	(*Inverter comm error*)	AddError[w_Index](
			b_ErrorTrig			:= Get.ui_InverterCommStatus <>0 AND Get.ui_InverterCommStatus <15, //general warning from inverter
			out_ST_Error			:= a_ActiveEvents[w_Index],
			w_ErrorID					:= 66 ,
			s_Message				:= 'inverter communication error',
			e_sev					:= eSeverity.Quickshutdown
			);
		IF AddError[w_Index].b_out THEN by_errCt := by_errCt + 1; END_IF;
		w_Index := w_Index +1;
		
	(*Inverter temp throttling active*)	AddError[w_Index](
			b_ErrorTrig			:= get.Events.b_TempThrottlingActive, //general warning from inverter
			out_ST_Error			:= a_ActiveEvents[w_Index],
			w_ErrorID					:= 67 ,
			s_Message				:= 'temperature throttling active',
			e_sev					:= eSeverity.Warning,
			b_AutoClear			:= TRUE,
			);
		IF AddError[w_Index].b_out THEN by_warnCt := by_warnCt + 1; END_IF;
		w_Index := w_Index +1;
		
	(*Inverter current throttling active*)	AddError[w_Index](
			b_ErrorTrig			:= get.Events.b_CurrThrottlingActive, //general warning from inverter
			out_ST_Error			:= a_ActiveEvents[w_Index],
			w_ErrorID					:= 68 ,
			s_Message				:= 'Current throttling active',
			e_sev					:= eSeverity.Warning,
			b_AutoClear			:= TRUE,
			);
		IF AddError[w_Index].b_out THEN by_warnCt := by_warnCt + 1; END_IF;
		w_Index := w_Index +1;
		
		(*Inverter current throttling active*)	AddError[w_Index](
			b_ErrorTrig			:= get.StatusWord.b_Fault, //general warning from inverter
			out_ST_Error			:= a_ActiveEvents[w_Index],
			w_ErrorID					:= 69,
			s_Message				:= 'General fault',
			e_sev					:= eSeverity.Quickshutdown,
			);
		IF AddError[w_Index].b_out THEN by_errCt := by_errCt + 1; END_IF;
		w_Index := w_Index +1;
		
		(*UVR fault*)			AddError[w_Index](
			b_ErrorTrig				:= Get.Events.b_24VdcUVRFault,
			out_ST_Error			:= a_ActiveEvents[w_Index],
			w_ErrorID				:= 70,
			s_Message				:= 'UVR 24VDC Fault',
			e_sev					:= eSeverity.warning,
			b_AutoClear				:= TRUE,
		);
		w_Index := w_Index +1;

			

get.events.b_GeneralFaultFlag := by_errCt <> 0;
get.events.b_GeneralWarningFlag := by_warnCt <>0;
END_METHOD

METHOD PRIVATE GetInverterModes
IF get.UgridStatusWord.b_AFEmodeActive THEN
	get.e_InverterMode := eInvertermodes.afe;
ELSIF get.UgridStatusWord.b_IslandModeActive OR get.UgridStatusWord.b_MicrogridModeActive AND get.r_FrequencyDroop <= 0.1 THEN
	get.e_InverterMode := eInvertermodes.Island;	
ELSE
	get.e_InverterMode := eInvertermodes.Microgrid;
END_IF
END_METHOD

METHOD PRIVATE GetMaxTemperature : REAL;
// calculate max
GetMaxTemperature := MAX(
						get.r_TemperatureCMChoke[1], 
						get.r_TemperatureCMChoke[2], 
						get.r_TemperatureCMChoke[3], 
						get.r_TemperatureCMChoke[4],
						get.r_TemperatureGridChoke[1], 
						get.r_TemperatureGridChoke[2], 
						get.r_TemperatureGridChoke[3]
);
END_METHOD

METHOD PRIVATE GetPowerModuleStatus : BOOL
IF get.StatusWord.b_Fault OR get.Events.b_GeneralFaultFlag THEN
	get.e_Status := eStatusPowerModule.fault;
ELSIF get.StatusWord.b_Running THEN
	get.e_Status := eStatusPowermodule.running;
ELSIF get.StatusWord.b_ReadyToOperate THEN
	get.e_Status := eStatusPowermodule.idle;
ELSIF get.StatusWord.b_DCAtReference THEN	
	get.e_Status := eStatusPowermodule.DcOK;
ELSIF get.StatusWord.b_ReadyToDCCharge THEN
	get.e_Status := eStatusPowermodule.off;
ELSE
	get.e_Status := eStatusPowermodule.Init;
END_IF
END_METHOD

METHOD GetTemperatureEvents : BOOL
VAR_INPUT
	Warnings	: 	BOOL;
END_VAR
IF Warnings THEN
	GetTemperatureEvents := get.Events.b_CMChokeTemperatureHigh[1] 	OR
			get.Events.b_CMChokeTemperatureHigh[2]		OR
			get.Events.b_CMChokeTemperatureHigh[3]		OR
			get.Events.b_CMChokeTemperatureHigh[4] 		OR
			get.Events.b_GridChokeTemperatureHigh[1]	OR
			get.Events.b_GridChokeTemperatureHigh[2]	OR
			get.Events.b_GridChokeTemperatureHigh[3]	OR
			get.Events.b_inverterTemperatureHigh;
ELSE
	GetTemperatureEvents := get.Events.b_CMChokeTemperatureTooHigh[1] 	OR
			get.Events.b_CMChokeTemperatureTooHigh[2]	OR
			get.Events.b_CMChokeTemperatureTooHigh[3]	OR
			get.Events.b_CMChokeTemperatureTooHigh[4]	OR
			get.Events.b_GridChokeTemperatureTooHigh[1]	OR
			get.Events.b_GridChokeTemperatureTooHigh[2]	OR
			get.Events.b_GridChokeTemperatureTooHigh[3]	OR
			get.Events.b_F56TemperatureFault;
END_IF
END_METHOD

METHOD Idle : BOOL
//Inverter.controlWord.b_ChargeDC := TRUE;
//inverter.ControlWord.b_run := TRUE;

//Set powermode
inverter.powermode := ePowermodes.Droop;
inverter.r_BaseCurrentRef := 0;
inverter.r_ReactiveCurrentRef := 0;
SetVoltageFrequency(SetToIn := TRUE, VoltIN := settings.GridParams.r_GridNominalVoltage, FreqIn := settings.GridParams.r_GridNominalFrequency);
inverter.startMode := FALSE;
inverter.Island(TRUE);
Idle := get.StatusWord.b_readytooperate AND NOT get.GridcodeStatusWord.b_GridCodeTripActive;

get.eConditioningRequirement := max(eConditioningRequirement.Pumprequired, ConditioningRequirement());
END_METHOD

METHOD init : BOOL

VAR_INST
	
END_VAR
inverter.ControlWord.b_ChargeDC := FALSE;
inverter.ControlWord.b_run := FALSE;
inverter.ControlWord.b_Reset := TRUE;
END_METHOD

METHOD Reset : BOOL
ton_ResetPulse(IN:= NOT ton_ResetPulse.Q);
set.b_QuickstopInactive := TRUE;

Inverter.ControlWord.b_Reset := TRUE;
buscoupler.b_MCCBChargeSpring := TRUE;

IF NOT (get.events.b_GeneralFaultFlag OR get.StatusWord.b_Fault) THEN
	Inverter.ControlWord.b_Reset := FALSE;
	buscoupler.b_MCCBChargeSpring := FALSE;
END_IF

ConditioningRequirement(true);
Reset := get.e_Status <> eStatusPowerModule.fault;
END_METHOD

METHOD Run : BOOL
VAR_INPUT
	Powermode			: ePowermodes;
	InverterMode		: EInvertermodes;
	InternalPowerSet		: BOOL;
END_VAR

VAR_INST
	r_DroopMin			: REAL;
	r_DroopMax			: REAL;
END_VAR
//Set powermodes
inverter.Powermode := powermode;
inverter.startMode := FALSE;

get.eConditioningRequirement := max(eConditioningRequirement.Pumprequired, ConditioningRequirement());

// set invertermode
CASE InverterMode OF
	eInverterModes.Afe : Inverter.AFE();
	eInverterModes.Microgrid : Inverter.Microgrid();
	eInverterModes.Island : Inverter.Island(FALSE);
END_CASE

SetVoltageFrequency(InternalPowerSet, set.r_NomVoltage, set.r_NomFrequency);

//Set absolute power and current limits of inverter
IF InternalPowerSet THEN
	inverter.r_InputActiveCurrentLimit := 100;
	inverter.r_OutputActiveCurrentLimit := 100;
	Inverter.Island(TRUE);
ELSE
	SetInverterRefs_Limits(get := get, set := set, 
		r_InputActiveCurrentLimitRef => inverter.r_InputActiveCurrentLimit,
		r_OutputActiveCurrentLimitRef => inverter.r_OutputActiveCurrentLimit,
		r_basecurrentref => inverter.r_BaseCurrentRef,
		r_ReactiveCurrentRef => inverter.r_ReactiveCurrentRef
	);
END_IF

inverter.ControlWord.b_run := TRUE;
run := get.StatusWord.b_Running;
END_METHOD

METHOD PRIVATE SetEvents
VAR_IN_OUT CONSTANT
	st_params					: ST_Powermodule_Params;
END_VAR


VAR_IN_OUT
	events						: ST_Powermodule_events;
END_VAR

VAR 
	w_Index										: WORD;
END_VAR

VAR_INST
	TempAnomalyThreshold	: REAL := 30;
	CMtempMediaan			: REAL;
	GridtempMediaan			: REAL;
	CMTempDeviation			: BOOL;
	GridTempDeviation		: BOOL;
END_VAR
//mediaan
CMtempMediaan := Median(get.r_TemperatureCMChoke);
GridtempMediaan := Median(get.r_TemperatureGridchoke);
CMTempDeviation := FALSE;
GridTempDeviation := FALSE;

FOR w_Index:=1 TO 4 DO
	IF ABS(get.r_TemperatureCMChoke[w_Index] - CMTempMediaan) > TempAnomalyThreshold THEN
		CMTempDeviation := TRUE;
	ELSE
	 LimitTrigger(
		r_IN := get.r_TemperatureCMChoke[w_Index],
		b_HighEnable:= TRUE,
		r_HighLimit:= st_Params.r_FilterTempAlarm,
		r_HighWarning:= st_params.r_FilterTempWarning,
		b_LowEnable:= FALSE,
		r_LowLimit:= 0,
		r_LowWarning:= 0,
		r_hysteresis:= 5,
		b_Warning=> get.Events.b_CMChokeTemperatureHigh[w_Index],
		b_Fault=> get.Events.b_CMChokeTemperatureTooHigh[w_Index]
		);
	END_IF
END_FOR

FOR w_Index:=1 TO 3 DO
	IF ABS(get.r_TemperatureGridChoke[w_Index] - GridTempMediaan) > TempAnomalyThreshold THEN
		GridTempDeviation := TRUE;
	ELSE
	LimitTrigger(
		r_IN := get.r_TemperatureGridChoke[w_Index],
		b_HighEnable:= TRUE,
		r_HighLimit:= st_params.r_FilterTempAlarm,
		r_HighWarning:= st_params.r_FilterTempWarning,
		b_LowEnable:= FALSE,
		r_LowLimit:= 0,
		r_LowWarning:= 0,
		r_hysteresis:= 5,
		b_Warning=>get.Events.b_GridChokeTemperatureHigh[w_Index],
		b_Fault=> get.Events.b_GridChokeTemperatureTooHigh[w_Index]
	);
	END_IF

END_FOR



// set warning when CMS PT100 gives out of range values. 
get.Events.b_CMSTemperatureRangeWarning := CMTempDeviation OR GridTempDeviation;

//Set fan state warning
get.Events.b_FanStateUnknownWarning := get.b_FanFb AND NOT buscoupler.b_FanOn;
get.Events.b_24VdcUVRFault := NOT get.b_MccbUvr24VdcOK AND get.b_DCcontactorFb;

//CMS average temperature
END_METHOD

METHOD PRIVATE SetInverterRefs_Limits : BOOL

VAR_IN_OUT
	get 			: ST_Powermodule_get;
	set				: ST_Powermodule_set;
END_VAR

VAR_OUTPUT
	r_InputActiveCurrentLimitRef : REAL;
	r_OutputActiveCurrentLimitRef : REAL;
	r_BaseCurrentRef			: REAL;
	r_ReactiveCurrentRef		: REAL;
END_VAR

VAR_INST
	r_PLimitOverhead				: REAL := 1.1;
	fb_ActiveCurrentMeasMA			: FB_movingAverage := (length := 1000, enable := TRUE);	
	r_MaxOvercurrentFactor			: REAL;	
	r_ActivePowerRQ					: REAL;
	r_ReactivePowerRQ				: REAL;
	fb_DynamicreactiveRemainMA		: FB_movingAverage := (length := 10, enable := TRUE);
	r_reactiveMaxCurrent			: REAL;
	r_ReactiveLimitCorrection		: REAL := 1.20;
	r_NomVoltage					: REAL := 400;
	ar_Throttling					: ARRAY [1..20] OF REAL;
	fb_SmoothThrottling				: FB_CTRL_Moving_Average := (eMode := e_ctrl_mode.eCTRL_MODE_ACTIVE);
	st_params_SmoothThrottling		: ST_CTRL_MOVING_AVERAGE_PARAMS := (
		 								tCtrlCycleTime := T#1S,
										tTaskCycleTime := T#1MS,
										nSamplesToFilter := 10);
										
	 r_InputActiveCurrentLimit		: REAL;
	 r_outputActiveCurrentLimit		: REAL;
	 r_baseCurrentSetpoint			: REAL;
	 r_reactiveCurrentsetpoint		: REAL;
	 r_VoltAC						: REAL;
	 r_DynamicCurrentLimit			: REAL;
	 r_ThrottlingValueFilterTemp	: REAL;
	 r_ThrottlingValueInverterTemp	: REAL;
	 r_ThrottlingValueMindex		: REAL;
	 r_ThrottlingActual				: REAL;
	 
	 
	 ePIDctrl						: E_CTRL_Mode;
	 //Mindex limiter
	r_ActReactiveToThrottlingValue	: REAL;
	fb_PIDMindex					: FB_CTRL_PID_EXT := (emode := e_Ctrl_mode.eCTRL_MODE_ACTIVE);
	st_Params_PIDMindex				: ST_CTRL_PID_EXT_PARAMS := ( 
										tTaskCycleTime := T#1MS,
										tCtrlCycleTime := T#1MS,
										fKp	:= 0.05,
										tTn := T#500MS,
										tTd := T#0S,
										tTv := T#0MS,
										fOutMaxLimit := 0,
										fOutMinLimit := -1,
										fouterwindow := 0
										);


	//AC current limiter
	fb_RampCurrentLimit				: FB_RAMP_Dual := (Enable := TRUE, rampDown := 50, rampUp := 20);									
	fb_PIDCurrentLimit				: FB_CTRL_PID_EXT;
	st_Params_PIDCurrentLimit		: ST_CTRL_PID_EXT_PARAMS := ( 
										tTaskCycleTime := T#1MS,
										tCtrlCycleTime := T#1MS,
										fKp	:= 0.5,
										tTn := T#500MS,
										tTd := T#0MS,
										tTv := T#0MS,
										fDeadbandInput := 10
										);
										
END_VAR
IF ton_ResetPulse.Q AND NOT get.StatusWord.b_Running THEN
	ePIDctrl := e_Ctrl_mode.eCTRL_MODE_RESET;
ELSE
	ePIDctrl := e_Ctrl_mode.eCTRL_MODE_Active;	
END_IF

r_VoltAC := get.r_ACVoltageSupply;
fb_ActiveCurrentMeasMA(IN := get.r_ActiveCurrent);
r_MaxOvercurrentFactor := MIN(st_params.r_ACCurrentLimitMax / MAX(1, st_params.r_InverterRatedCurrent), set.r_overcurrentFactor);

st_params_SmoothThrottling.pWorkArray_ADR := ADR(ar_Throttling);
st_params_SmoothThrottling.nWorkArray_SIZEOF := SIZEOF(ar_Throttling);

fb_SmoothThrottling(
	fin := get.r_TemperatureMax,
	stParams := st_params_SmoothThrottling);

r_ThrottlingValueFilterTemp := scale(
		r_in:=fb_SmoothThrottling.fOut,
		 In_min:= st_params.r_FilterTempWarning,
		 In_max:= st_params.r_FilterTempAlarm,
		 Out_min:= r_MaxOvercurrentFactor,
		 Out_max:= st_params.r_ThrottlingMinimum);
		
r_ThrottlingValueInverterTemp := scale(
		r_in:=get.r_TemperatureInverter,
		 In_min:= st_params.r_InverterTempWarning,
		 In_max:= st_params.r_InverterTempAlarm,
		 Out_min:= r_MaxOvercurrentFactor,
		 Out_max:= st_params.r_ThrottlingMinimum);	

r_ThrottlingActual	:= MIN(r_ThrottlingValueInverterTemp,r_ThrottlingValueFilterTemp);	

//TOTAL AC CURRENT LIMIT
	st_Params_PIDCurrentLimit.fOutMaxLimit := st_params.r_ACCurrentLimitMax;
	st_Params_PIDCurrentLimit.fOutMinLimit := st_params.r_ACCurrentLimitMin;
	fb_RampCurrentLimit(SetToIn := NOT get.StatusWord.b_Running, IN :=  LIMIT(st_params.r_ACcurrentLimitMin, set.r_ACcurrentLimit, st_params.r_InverterRatedCurrent *  r_throttlingActual));
	fb_PIDCurrentLimit(
		eMode := ePIDctrl,
		fSetpointValue := LIMIT(fb_RampCurrentLimit.Q,get.r_ACCurrent, fb_RampCurrentLimit.Q),
		fActualValue := get.r_ACCurrent,
		stParams:= st_params_PIDCurrentLimit,
		fout => r_DynamicCurrentLimit
		);
	
	IF fb_PIDCurrentLimit.bError THEN
		r_DynamicCurrentLimit := LIMIT(st_params.r_ACcurrentLimitMin, set.r_ACcurrentLimit, st_params.r_InverterRatedCurrent *  r_throttlingActual);
	END_IF
	
	IF st_calibration.b_StartCalibration THEN
		r_DynamicCurrentLimit := 650;
	END_IF

//ACTIVE CURRENT LIMIT
	r_InputActiveCurrentLimit := LIMIT(0 , kWToCurrent(ABS(set.r_Pmin), 400), st_params.r_ACCurrentLimitMax);
	r_OutputActiveCurrentLimit := LIMIT(0 , kWToCurrent(ABS(set.r_Pmax),  400), st_params.r_ACCurrentLimitMax);

//ACTIVE SETPOINT
	r_activePowerRQ := CompensationCurve(PIN := set.r_ActivePower, QIN := get.r_ReactivePower, coef := st_calibration.PCoefficients, mode := 0);
	r_ActivePowerRQ	:= LIMIT(get.r_Pmin, r_ActivePowerRQ, get.r_Pmax);


//REACTIVE SETPOINT + MINDEX LIMIT
st_params_PIDMindex.fDeadBandInput := st_params.r_ModulationIndexLimitHyst;
	fb_PIDMindex(
		eMode := ePIDctrl,
		fsetpointvalue :=  st_params.r_ModulationIndexLimit,
		fActualValue := get.r_ModulationIndex,
		stparams := st_Params_PIDMindex
	);	
	r_ThrottlingValueMindex := fb_PIDMindex.fout + 1;
	fb_DynamicreactiveRemainMA(IN := SQRT(MAX(EXPT(r_DynamicCurrentLimit,2) - EXPT(fb_ActiveCurrentMeasMA.Q*r_ReactiveLimitCorrection ,2), 0)) * r_ThrottlingValueMindex);
	r_ReactivePowerRQ := CompensationCurve(PIN := get.r_activePower, QIN := set.r_ReactivePower, coef := st_calibration.QCoefficients, mode := 1);
	
	//to jump to PID value when throttling starts. Otherwise takes quite some time to get there.
	r_ActReactiveToThrottlingValue := kWToCurrent(r_ActivePowerRQ, get.r_ACVoltageD7) / MAX(1, fb_DynamicreactiveRemainMA.Q);
	IF get.r_ModulationIndex > MIN(100, st_params.r_ModulationIndexLimit + st_params.r_ModulationIndexLimitHyst) AND r_ThrottlingValueMindex > r_ActReactiveToThrottlingValue THEN
		fb_PIDMindex.fManSyncValue := r_ActReactiveToThrottlingValue - 1;
		fb_PIDMindex.bSync := TRUE;
	ELSE
		fb_PIDMindex.bSync := FALSE;
	END_IF
	
//power overwrites before it is converted to refs
	IF st_calibration.b_StartCalibration THEN
		r_activePowerRQ := st_calibration.r_Pset;
		r_ReactivePowerRQ	:= st_calibration.r_Qset;
	END_IF

//To currents
	r_basecurrentSetpoint := LIMIT(-r_DynamicCurrentLimit, kWToCurrent(r_ActivePowerRQ, r_VoltAC), r_DynamicCurrentLimit);
	r_reactiveCurrentSetpoint := LIMIT(-fb_DynamicreactiveRemainMA.Q, kWToCurrent(r_ReactivePowerRQ,get.r_ACVoltageD7), fb_DynamicreactiveRemainMA.Q);	

//TO REFS
	r_InputActiveCurrentLimitRef := BaseValueToRef(r_InputActiveCurrentLimit);
	r_OutputActiveCurrentLimitRef := BaseValueToRef(r_OutputActiveCurrentLimit);
	r_baseCurrentRef := BaseValueToRef(r_basecurrentSetpoint);
	r_ReactivecurrentRef:= BaseValueToRef(r_reactiveCurrentSetpoint);

get.b_LimiterActive := TRUE;
// set limter state
IF r_ThrottlingValueMindex < fb_PIDMindex.fManSyncValue THEN
	get.e_ThrottlingStatus := ePowerModuleThrottlingState.Overvoltage;
ELSIF r_ThrottlingValueFilterTemp < r_MaxOvercurrentFactor THEN
	get.e_ThrottlingStatus := ePowerModuleThrottlingState.FilterTemp;
ELSIF r_ThrottlingValueInverterTemp < r_MaxOvercurrentFactor THEN
	get.e_ThrottlingStatus := ePowerModuleThrottlingState.InverterTemp;
ELSE
	get.b_LimiterActive := FALSE;
END_IF


	
//set the final value as feedback to the get struct of the powermodule
	get.r_OverCurrentValue 	:=  r_ThrottlingActual;
	get.r_Pmin 				:= -CurrentToKw(MIN(get.r_ACcurrentLimit, r_InputActiveCurrentLimit), r_VoltAC) * r_PLimitOverhead;
	get.r_Pmax 				:= CurrentToKw(MIN(get.r_ACcurrentLimit, r_outputActiveCurrentLimit), r_VoltAC);
	get.r_ACcurrentLimit	:= MIN(set.r_ACcurrentLimit, r_DynamicCurrentLimit);
	r_reactiveMaxCurrent 	:= MIN(fb_DynamicreactiveRemainMA.Q, SQRT(MAX(EXPT(get.r_ACcurrentLimit,2) - EXPT(get.r_ActiveCurrent,2), 0)));
	get.r_Qmax				:=  CurrentToKW(r_reactiveMaxCurrent, r_VoltAC);
	get.r_Qmin				:= -get.r_Qmax;
END_METHOD

METHOD PRIVATE SetInverterSettings : BOOL

VAR_INST
	ton_GridcodeOnDelay	: TON := (PT:= T#500MS);
	ton_GridcodeOffDelay: TON := (PT:= T#0S);
	SR_GridCodeActivate	: SR; 
	
	FtrigResetDrive		: F_TRIG;
END_VAR
//set actual droop
inverter.r_BaseRefRampRate		:= set.i_PowerChangeRate;

ton_GridcodeOffDelay(IN := (get.e_InverterMode <> eInvertermodes.Afe AND NOT get.GridcodeStatusWord.b_GridCodeTripActive) OR NOT get.StatusWord.b_Running);
ton_GridcodeOnDelay(IN:= get.e_InverterMode = eInvertermodes.Afe AND set.b_gridcodeEnable AND get.StatusWord.b_ReadyToOperate);
//Set gridcodes
SR_GridCodeActivate(
	SET1 := ton_GridcodeOnDelay.Q,
	RESET := ton_GridcodeOffDelay.Q OR NOT set.b_gridcodeEnable OR NOT get.StatusWord.b_ReadyToOperate,
	);


inverter.ControlWord.b_GridCodeEnable:= SR_GridCodeActivate.Q1;
inverter.controlword.b_ExtGridcodeTrip := set.b_ExtgridCodeTrip;

//reset drive if gridcodes are set off
FtrigResetDrive(CLK:= inverter.ControlWord.b_GridCodeEnable);
IF FtrigResetDrive.Q THEN
	Reset();
END_IF

IF NOT get.StatusWord.b_Running THEN
	//Set powermode
	inverter.Island(TRUE);
	//Set voltage / frequency
	//SetVoltageFrequency(TRUE, settings.GridParams.r_GridNominalVoltage, settings.GridParams.r_GridNominalFrequency);	
END_IF
END_METHOD

METHOD PRIVATE SetParallelDrive : BOOL
IF Settings.Configuration.b_DoublePowerModule THEN
	inverter.ControlWord.b_ParallelAFE := TRUE;
ELSE
	inverter.ControlWord.b_ParallelAFE:= FALSE;
END_IF

SetParallelDrive := Settings.Configuration.b_DoublePowerModule;
END_METHOD

METHOD SetVoltageFrequency : BOOL
VAR_INPUT
	SetToIn		: BOOL;
	VoltIN		: REAL;
	FreqIN		: REAL;
END_VAR

VAR_INST
	//rTrig_SetToIN	: R_TRIG;
END_VAR

VAR_INST
	r_FrequencyDroopOffset 	: REAL;
	r_VoltageDroopOffset 	: REAL;
	//freqRamp				: FB_ramp := (b_enable := TRUE, r_rampRate := 10);
	//VoltRamp				: FB_ramp := (b_enable := TRUE, r_rampRate := 10);
END_VAR
//rTrig_SetToIN(CLK := SetToIn);
//FreqRamp(SetToIn := NOT get.StatusWord.b_Running OR rTrig_SetToIN.Q);
//VoltRamp(SetToIn := NOT get.StatusWord.b_Running OR rTrig_SetToIN.Q);
//FreqRamp.IN := FreqIN;	
//VoltRamp.IN := VoltIN;

// set gridnominal Frequency
r_FrequencyDroopOffset := FreqIN - settings.GridParams.r_GridNominalFrequency;
inverter.r_FrequencyDroopOffset := LIMIT(-2, r_FrequencyDroopOffset, 2);
// set gridnominal voltage
r_VoltageDroopOffset := VoltIN - settings.GridParams.r_GridNominalVoltage + st_params.i_VoltageOffset;
inverter.r_VoltageCorrection	:= LIMIT(-40 + st_params.i_VoltageOffset, r_VoltageDroopOffset, 40 + st_params.i_VoltageOffset);
END_METHOD

METHOD Shutdown : BOOL
VAR_INPUT
	b_Force		: BOOL := FALSE;
END_VAR

VAR_INST
	b_enableForce : BOOL := FALSE;
	currentMax : REAL;
	r_DCcurrentAbs : REAL;
	r_DCcurrent	: REAL;
END_VAR

VAR
	r_DCreleaseCurrent		: REAL := 20;
END_VAR
r_DCcurrentAbs := ABS(get.r_DCCurrent);
inverter.r_BaseCurrentRef := 0;
inverter.r_ReactiveCurrentRef := 0;

IF (b_Force OR get.StatusWord.b_Fault) THEN
	inverter.ControlWord.b_ChargeDC := FALSE;
	inverter.ControlWord.b_run := FALSE;
ELSE
	inverter.ControlWord.b_run := FALSE;
	inverter.r_OutputActiveCurrentLimit := 10;
	inverter.r_InputActiveCurrentLimit := 10;
	IF r_DCcurrentAbs < r_DCreleaseCurrent THEN
		inverter.ControlWord.b_ChargeDC := FALSE;
		buscoupler.b_MCCBChargeSpring := TRUE;	
	END_IF
END_IF

ConditioningRequirement(true);
get.eConditioningRequirement := eConditioningrequirement.none;

//minimum shutdown execution time.
shutdown := NOT inverter.ControlWord.b_ChargeDC AND NOT inverter.ControlWord.b_run AND NOT get.StatusWord.b_Running AND DecoupleDC();
END_METHOD

METHOD Start : BOOL

VAR_INPUT
	AFESTART : BOOL;
END_VAR

VAR_INST
	tp_RunDelay			: TP := (PT:= T#1S);
	StartupValue		:	BOOL := TRUE;
	b_RunAlready		: BOOl;
END_VAR
inverter.r_OutputActiveCurrentLimit := 520;
inverter.r_InputActiveCurrentLimit := 520; 
inverter.ControlWord.b_run := FALSE;
inverter.startMode := TRUE;

IF AFESTART THEN
	inverter.AFE();
ELSE
	inverter.Island(TRUE);
END_IF

SetVoltageFrequency(TRUE, settings.GridParams.r_GridNominalVoltage, settings.GridParams.r_GridNominalFrequency);

(*STEPS
first check if DC exists
if its yet there and checkDCvoltage gives TRUE, inverter can get to run state.
Ifnot, try precharging (if its in the system).

*)
IF get.b_MccbUvr24VdcOK THEN
	inverter.ControlWord.b_ChargeDC := get.StatusWord.b_ReadyToDCCharge;
	tp_RunDelay(in := CheckDCvoltage() AND NOT tp_RunDelay.Q);
	b_RunAlready := get.StatusWord.b_running AND get.r_ACVoltageSupply <> 0;
	inverter.ControlWord.b_run := tp_RunDelay.Q OR b_RunAlready;
END_IF


//Check if we already have DC
IF CoupleDC() THEN
	Start := get.StatusWord.b_Running;
END_IF

get.eConditioningRequirement := eConditioningrequirement.none;



//OLD code, run delay and startup value might be needed -- To be tested
(*


IF CheckDCvoltage(r_BatDcVoltage) THEN
	inverter.ControlWord.b_ChargeDC := get.StatusWord.b_ReadyToDCCharge;
	inverter.ControlWord.b_run := tp_RunDelay.Q OR startupValue;
	StartupValue := FALSE;
	
	IF get.StatusWord.b_Running THEN
		tp_RunDelay(in := FALSE);
	END_IF
	Start := get.StatusWord.b_Running;
END_IF
*)
END_METHOD

END_FUNCTION_BLOCK

// ---- POUs/Objects/PowerStack/PowerModule/FB_PowerModule_Inverter.TcPOU
FUNCTION_BLOCK FB_PowerModule_Inverter
VAR_IN_OUT
	get									: ST_PowerModule_Get;
	set									: ST_Powermodule_Set;
END_VAR

VAR_IN_OUT CONSTANT
	st_params							: ST_PowerModule_params;									
END_VAR

VAR_INPUT
	b_parallelDrive						: BOOL;
	ControlWord							: ST_InverterControlWord;
	r_InputActiveCurrentLimit			: REAL;
	r_OutputActiveCurrentLimit			: REAL;
	
//current refs for power calc
	r_BaseCurrentRef					: REAL;
	r_BaseRefRampRate					: REAL;
	r_ReactiveCurrentRef				: REAL;
	r_FrequencyDroopOffset				: REAL;
	r_VoltageCorrection					: REAL;
	Powermode							: ePowermodes;
	StartMode							: BOOL;
END_VAR	

VAR
	// Local variables
	//IO variables
	a_StatusDataIN					AT %I* : ARRAY[1..2] OF UINT;
	a_ProcessDataIN					AT %I* : ARRAY[1..16] OF INT;
	a_ControlDataOUT				AT %Q* : ARRAY[1..1] OF UINT;
	a_ProcessDataOUT				AT %Q* : ARRAY[1..16] OF INT;
	
	i_InverterMode					: INT; // 0= AFE, 1= ugrid	
END_VAR

VAR_STAT
	r_DroopMax						: REAL;
	r_DroopMin						: REAL;
	r_DroopIsland					: REAL;
	
	//Power mode final
	w_StartPowerMode				: WORD;  // 0= Zero D7, 1= Zero Supply, 2= Droop, 3= iso
	w_StartVoltageMode				: WORD;	// 0= Zero D7, 1= Droop, 2= Keep reactive Ref (iso)
END_VAR


// Read data
Read();

//Watchdog Feedback and pulse
WatchdogTimer();

//Setpowermode
SetPowermode();

//Write data
Write(get, st_params);

METHOD AFE : BOOL
VAR_INPUT
END_VAR
i_invertermode	:= 0; //AFE
r_DroopMin := set.r_DroopMaximum;
r_DroopMax := set.r_DroopMaximum;
END_METHOD

METHOD PRIVATE IntPercentageToReal : REAL
VAR_INPUT
	in				: INT;
	ratedCurrent	: REAL;
END_VAR
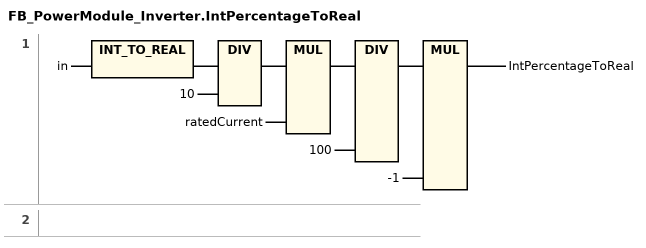
// NETWORK 1
IntPercentageToReal := (((INT_TO_REAL(in) / 10) * ratedCurrent) / 100) * -1;

// NETWORK 2
END_METHOD

METHOD Island : BOOL
VAR_INPUT
	soft	: BOOL;
END_VAR
i_invertermode := 2; //Ugrid
r_DroopMin:= set.r_DroopIslandMode;
r_DroopMax:= set.r_DroopIslandMode;


IF soft THEN
	powermode := ePowermodes.DroopZeroStart;
	r_DroopMin:= 1;
	r_DroopMax:= 1;
ELSE
	powermode := ePowermodes.Droop;
	r_DroopMin:= set.r_DroopIslandMode;
	r_DroopMax:= set.r_DroopIslandMode;
END_IF
END_METHOD

METHOD Microgrid : BOOL

VAR_INPUT
	
END_VAR
i_invertermode := 2; //Ugrid
r_DroopMin := set.r_DroopMinimum;
r_DroopMax := set.r_DroopMaximum;
END_METHOD

METHOD Read : BOOL

VAR_INST
	w_MicrogridStatusWord		: WORD;
	w_FaultStatusWord1			: WORD;
	w_FaultStatusWord2			: WORD;
	w_GridcodeStatusWord		: WORD;
	w_ModulationIndex			: WORD;
	ModulationIndexMA			: fb_MovingAverage := (enable := TRUE,  length:= 100);
END_VAR
//Convert get.RawReadData to right data type and range.
	w_MicrogridStatusWord		:= TO_WORD(a_ProcessDataIn[1]); 
	get.r_DCVoltage 			:= INT_TO_REAL(a_ProcessDataIn[2]);
	get.r_DCCurrent				:= -INT_TO_REAL(a_ProcessDataIn[3]);
	get.r_D7SyncError			:= scale(r_in:= INT_TO_REAL(a_ProcessDataIn[4]), In_min :=-3072, In_max:=3071, Out_min:=-180, Out_max:= 180);
	get.r_ActiveCurrent			:= IntPercentageToReal(a_ProcessDataIn[5], st_params.r_InverterRatedCurrent);
	get.r_ReactiveCurrent		:= IntPercentageToReal(a_ProcessDataIn[6], st_params.r_InverterRatedCurrent);
	get.r_ACVoltageD7			:= INT_TO_REAL(a_ProcessDataIn[7]);
	get.r_FrequencyD7			:= MAX(0, INT_TO_REAL(a_ProcessDataIn[8]))/100;
	get.r_TemperatureInverter	:= INT_TO_REAL(a_ProcessDataIn[9]);
	get.r_ACVoltageSupply		:= INT_TO_REAL(a_ProcessDataIn[10])/10;
	get.r_FrequencySupply		:= MAX(0, INT_TO_REAL(a_ProcessDataIn[11]))/100;
	get.r_ACCurrent				:= INT_TO_REAL(a_ProcessDataIn[12]);
	w_FaultStatusWord1			:= TO_WORD(a_ProcessDataIn[13]);
	w_FaultStatusWord2			:= TO_WORD(a_ProcessDataIn[14]);
	w_GridcodeStatusWord		:= TO_WORD(a_processDataIN[15]);
	w_modulationIndex			:= TO_WORD(a_processDataIN[16]);

ModulationIndexMA(IN := TO_REAL(w_modulationIndex)/ 10, Q => get.r_ModulationIndex);

//UNPACK General Status Word
UnpackWord(
	w_IN:= TO_WORD(a_StatusDataIn[1]),
	b0=>get.StatusWord.b_ReadyToDCCharge,
	b1=>get.StatusWord.b_ReadyToOperate,
	b2=>get.StatusWord.b_Running,
	b3=>get.StatusWord.b_Fault,
	b4=>get.StatusWord.b_RunEnabled,
	b5=>get.StatusWord.b_QuickstopNotActive,
	b6=>get.StatusWord.b_MCCBControlNotOK,
	b7=>get.StatusWord.b_Warning,
	b8=>get.StatusWord.b_DCAtReference,
	b9=>,
	b10=>get.StatusWord.b_DCAboveLimit,
	b11=>,
	b12=>,
	b13=>,
	b14=>,
	b15=>get.StatusWord.b_WatchdogFeedback,
);

get.ui_InverterCommStatus := a_StatusDataIn[2];

//UNPACK Ugridword 
UnpackWord(
	w_IN:= w_MicrogridStatusword,
	b0=>Get.UgridStatusWord.b_ChargeControlActive,
	b1=>get.UgridStatusWord.b_InternalChargingSwitchStatus,
	b2=>get.UgridStatusWord.b_MCBcontrol,
	b3=>Get.UgridStatusWord.b_MCBStatus,
	b4=>Get.UgridStatusWord.b_RunEnabled,
	b5=>Get.UgridStatusWord.b_DriveReady,
	b6=>Get.UgridStatusWord.b_AFEmodeActive,
	b7=>Get.UgridStatusWord.b_IslandModeActive,
	b8=>Get.UgridStatusWord.b_MicrogridModeActive,
	b9=>Get.UgridStatusWord.b_RunRequestActive,
	b10=>Get.UgridStatusWord.b_DriveInRunState,
	b11=>Get.UgridStatusWord.b_FaultActive,
	b12=>Get.UgridStatusWord.b_SynchronizedToD7,
	b13=>,
	b14=>Get.UgridStatusWord.b_D7MeasurementsOK,
	b15=>
);

//get mccbfb from inverter ugrid word.
Get.b_MccbFb := get.UgridStatusWord.b_MCBStatus;

//UNPACK Fault Word
UnpackWord(
	w_IN:= w_FaultStatusWord1,
	b0=>get.Events.b_F1OverCurrent,
	b1=>get.Events.b_F2OverVoltage,
	b2=>get.Events.b_F9UnderVoltage,
	b3=>get.Events.b_F91ShortCircuit,
	b4=>get.Events.b_F3EarthFault,
	b5=>,
	b6=>get.Events.b_F14UnitOverTemperature,
	b7=>get.Events.b_F56TemperatureFault,
	b8=>get.Events.b_F10LineSynchFault,
	b9=>,
	b10=>,
	b11=>get.Events.b_F52KeypadOCCommFault,
	b12=>get.Events.b_F53FieldbusFault,
	b13=>get.Events.b_F59SystembusFault,
	b14=>get.Events.b_F54SlotCommunicationFault,
	b15=>get.Events.b_F50Meas4mAFault
);

UnpackWord(
	w_IN:= w_FaultStatusWord2,
	b0=>get.Events.b_F11OutputPhaseFault,
	b1=>get.Events.b_F80ChargeFault,
	b2=>,
	b3=>,
	b4=>,
	b5=>,
	b6=>get.Events.b_F51ExternalFault,
	b7=>,
	b8=>,
	b9=>get.Events.b_F31IGBTFault,
	b10=>,
	b11=>,
	b12=>,
	b13=>,
	b14=>get.Events.b_F64MCBstateFault,
	b15=>
);

UnpackWord(
	w_IN:= w_GridcodeStatusWord,
	b0=>get.GridcodeStatusWord.b_LineVoltTripLimHigh,
	b1=>get.GridcodeStatusWord.b_LineVoltTripLimLow,
	b2=>get.GridcodeStatusWord.b_LineFreqTripLimHigh,
	b3=>get.GridcodeStatusWord.b_LineFreqTripLimLow,
	b4=>,
	b5=>,
	b6=>,
	b7=>,
	b8=>,
	b9=>,
	b10=>,
	b11=>get.GridcodeStatusWord.b_LineFreqOK,
	b12=>get.GridcodeStatusWord.b_LineVoltOK,
	b13=>get.GridcodeStatusWord.b_FRTActive,
	b14=>,
	b15=>get.GridcodeStatusWord.b_GridCodeTripActive
);


(*
INFO VACON IDs

Status word				: ID68, see ARFIF106 manual
1.Line state word		: ID3547,  (gridcode state) --> shift down
1.MicroGridSW			: ID1701, see ARFIF106 manual
2.DCVoltage				: ID1108, unit: VDC
3.DCCurrent				: ID72, Unit: Ampere DC
4.D7 Sync Error 		: ID1659, Unit: degree -3072...+3071 = -180...180 degrees.
5.ActiveCurrent			: ID1125, Unit: % of rated current
6.ReactiveCurrent 		: ID1157, Unit: % of rated current 
7.Line Voltage D7		: ID1650, Unit: VAC
8.Frequency D7			: ID1654, Unit: Hz
9.Unit temperature		: ID1109, Unit: C
10.Line voltage Supply	: ID1107, Unit: VAC
11.Frequency Supply		: ID1	, Unit: Hz
12.Total current 		: ID1104, Unit: A
13.
14.Fault Word 1		: ID1172, See ARFIF106 manual
15. 
16.

*)
END_METHOD

METHOD PRIVATE RealToInt : INT
VAR_INPUT
	in_r_Value				: REAL ;
	in_r_Res				: REAL ;
	in_i_Offset				: INT ;
END_VAR
VAR
	r_ResolutionResolved	: REAL;
	r_OffsetSolved			: REAL;
END_VAR
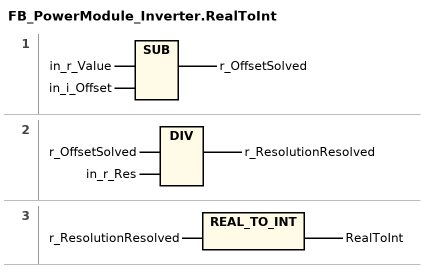
// NETWORK 1
r_OffsetSolved := in_r_Value - in_i_Offset;

// NETWORK 2
r_ResolutionResolved := r_OffsetSolved / in_r_Res;

// NETWORK 3
RealToInt := REAL_TO_INT(r_ResolutionResolved);
END_METHOD

METHOD PRIVATE SetPowerMode : BOOL
// SET Powermodes
CASE Powermode OF
	ePowermodes.DroopZeroStart : 
		get.e_PowerMode			:= ePowerModes.DroopZeroStart;
		w_StartPowerMode		:= 0;
		w_StartVoltageMode		:= 0;
	ePowermodes.Droop :
		get.e_PowerMode			:= ePowerModes.Droop;
		w_StartPowerMode		:= 2;
		w_StartVoltageMode		:= 1;
	ePowermodes.Isochronous :
		get.e_PowerMode			:= ePowerModes.Isochronous;
		w_StartPowerMode		:= 3;
		w_StartVoltageMode		:= 2;
END_CASE

IF startmode THEN
	get.e_PowerMode			:= ePowerModes.DroopZeroStart;
	w_StartPowerMode		:= 0;
	w_StartVoltageMode		:= 0;
END_IF
END_METHOD

METHOD PRIVATE UnpackWord : BOOL
VAR_INPUT
	w_IN			: WORD;
END_VAR

VAR_OUTPUT
	b0			: BOOL;
	b1			: BOOL;
	b2			: BOOL;
	b3			: BOOL;
	b4			: BOOL;
	b5			: BOOL;
	b6			: BOOL;
	b7			: BOOL;
	b8			: BOOL;
	b9			: BOOL;
	b10			: BOOL;
	b11			: BOOL;
	b12			: BOOL;
	b13			: BOOL;
	b14			: BOOL;
	b15			: BOOL;
END_VAR
b0 := w_IN.0;
b1 := w_IN.1;
b2 := w_IN.2;
b3 := w_IN.3;
b4 := w_IN.4;
b5 := w_IN.5;
b6 := w_IN.6;
b7 := w_IN.7;
b8 := w_IN.8;
b9 := w_IN.9;
b10 := w_IN.10;
b11 := w_IN.11;
b12 := w_IN.12;
b13 := w_IN.13;
b14 := w_IN.14;
b15 := w_IN.15;
END_METHOD

METHOD PRIVATE WatchdogTimer : BOOL 

VAR_INST
	t_WatchdogFb1				: TON;
	t_WatchdogFB2				: TON;
	t_WatchdogTimer1			: TON;
	t_WatchdogTimer2			: TON;
	b_WatchdogPulseFalse		: BOOL;
END_VAR
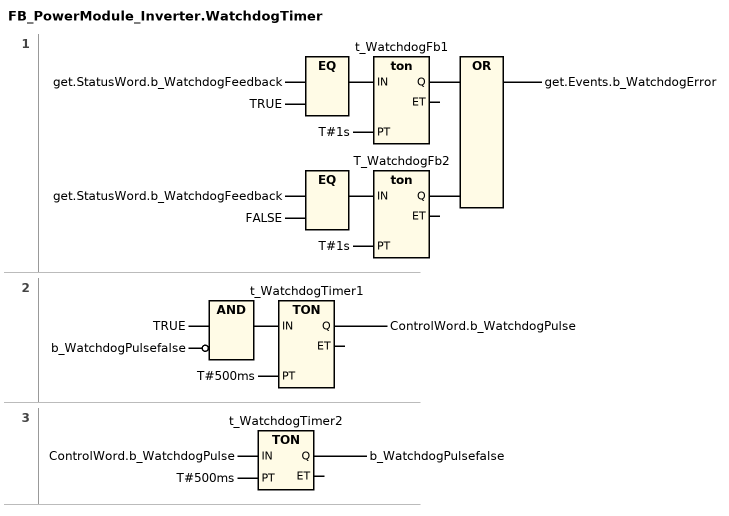
// NETWORK 1
t_WatchdogFb1(IN := get.StatusWord.b_WatchdogFeedback = TRUE, PT := T#1s); // ton
T_WatchdogFb2(IN := get.StatusWord.b_WatchdogFeedback = FALSE, PT := T#1s); // ton
get.Events.b_WatchdogError := t_WatchdogFb1.Q OR T_WatchdogFb2.Q;

// NETWORK 2
t_WatchdogTimer1(IN := TRUE AND NOT b_WatchdogPulsefalse, PT := T#500ms); // TON
ControlWord.b_WatchdogPulse := t_WatchdogTimer1.Q;

// NETWORK 3
t_WatchdogTimer2(IN := ControlWord.b_WatchdogPulse, PT := T#500ms); // TON
b_WatchdogPulsefalse := t_WatchdogTimer2.Q;
END_METHOD

METHOD Write : BOOL
VAR_IN_OUT
	get : ST_Powermodule_get;
END_VAR

VAR_IN_OUT CONSTANT
	st_params							: ST_PowerModule_params;									
END_VAR

VAR_INST
	b_rampEnable						: BOOL := TRUE;		
	fb_Ramp_OutactLim					: FB_Ramp := (r_RampRate:=100);
	fb_Ramp_InActLim					: FB_Ramp := (r_RampRate:=100);	
	
	r_FreqDroopAct						: REAL;
	r_VoltDroopAct						: REAL;
END_VAR
fb_Ramp_OutActLim(IN:=r_OutputActiveCurrentLimit, b_enable:= b_rampEnable);
fb_Ramp_InActLim(IN:=r_InputActiveCurrentLimit, b_enable:= b_rampEnable);

IF get.e_PowerMode = ePowerModes.Isochronous OR startmode THEN
	r_FreqDroopAct := set.r_DroopMaximum;
	r_VoltDroopAct := set.r_DroopMaximum;
ELSE
	r_FreqDroopAct := LIMIT(r_DroopMin, set.r_FrequencyDroop, r_DroopMax);
	r_VoltDroopAct := LIMIT(r_DroopMin, set.r_VoltageDroop, r_DroopMax);
END_IF

//get
get.controldata.Controlword := controlword;
get.controldata.i_invertermode := i_invertermode;
get.controldata.i_BaseCurrentRef := RealToInt(r_BaseCurrentRef, 0.1, 0);
get.controldata.i_ReactiveCurrentRef:= RealToInt(-r_ReactiveCurrentRef, 0.1, 0);
get.controldata.i_FrequencyDroop := RealToInt(r_FreqDroopAct , 0.002, 0); // Convert percentage to  mHz and rescale. So +100% ==> +5000.0 mHz
get.controldata.i_VoltageDroop := RealToInt(r_VoltDroopAct, 0.01, 0);
get.controldata.i_FrequencyDroopOffset := RealToInt(r_FrequencyDroopOffset, 0.01, 0);
get.controldata.i_VoltageCorrection := RealToInt(r_VoltageCorrection, 1, 0);
get.controldata.i_BaseRefRampRate := LIMIT(-1, RealToInt(r_BaseRefRampRate, 1, 0),10000);
get.controldata.i_StartPowerMode := WORD_TO_INT(w_StartPowerMode);
get.controldata.i_StartVoltageMode := WORD_TO_INT(w_StartVoltageMode);
get.controldata.i_OutActCurrentLimit := RealToInt(fb_Ramp_OutActLim.Q, 0.1, 0);
get.controldata.i_InActCurrentLimit := RealToInt(fb_Ramp_InActLim.Q, 0.1, 0);
get.controldata.i_DCVramprate :=  LIMIT(-1, st_params.i_DCVramprate, 10000);
get.r_FrequencyDroop := r_FreqDroopAct;
get.r_VoltageDroop := r_VoltDroopAct;



get.controldata.ui_controlwordvalue	:= PackWord(
	b0:=ControlWord.b_ChargeDC,
	b1:= TRUE, //b_MccbCloseEnable,
	b2:= TRUE,//set.b_QuickstopInactive,
	b3:= SEL(set.b_RunEnable, FALSE, ControlWord.b_Run),
	b4:=TRUE, //b_OutputpowerLimits,
	b5:=TRUE, //b_PowerIncreaseEnable,
	b6:=TRUE,//b_InputpowerLimits,
	b7:= ControlWord.b_Reset,
	b8:=0,
	b9:=0,
	b10:= ControlWord.b_FieldbusControlEnable,
	b11:= ControlWord.b_WatchdogPulse,
	b12:= ControlWord.b_ParallelAFE, // ID1501
	b13:= ControlWord.b_GridCodeEnable,
	b14:= ControlWord.b_ExtGridcodeTrip, // ID3310
	b15:=0
);

a_ControlDataOUT[1]	:= get.controldata.ui_controlwordvalue;
a_ProcessDataOUT[1] := get.controldata.i_invertermode;
a_ProcessDataOUT[2] := get.controldata.i_BaseCurrentRef;
a_ProcessDataOUT[3] := get.controldata.i_ReactiveCurrentRef;
a_ProcessDataOUT[4]	:= get.controldata.i_FrequencyDroop;
a_ProcessDataOUT[5]	:= get.controldata.i_VoltageDroop;
a_ProcessDataOUT[6]	:= get.controldata.i_FrequencyDroopOffset;
a_ProcessDataOUT[7]	:= get.controldata.i_VoltageCorrection;
a_ProcessDataOUT[8]	:= get.controldata.i_BaseRefRampRate;
a_ProcessDataOUT[9]	:= get.controldata.i_StartPowerMode;
a_ProcessDataOUT[10]:= get.controldata.i_StartVoltageMode;
a_ProcessDataOUT[11]:= get.controldata.i_OutActCurrentLimit;
a_ProcessDataOUT[12]:= get.controldata.i_InActCurrentLimit;
a_ProcessDataOUT[13]:= get.controldata.i_DCVramprate;
//a_ProcessDataOUT[14]	:= RESERVE;
//a_ProcessDataOUT[15]	:= RESERVE;
//a_ProcessDataOUT[16]	:= RESERVE;

(*
INVERTER CONTROLS:
FBFixedCW				: ID1160, Vacon AFE 2 Profile (3) to be set in NCDRIVE
1.ControlMode				: ID1531, 0: AFE, 1: Ugrid, 2: Island
2.BaseCurrentReference		: ID1533, unit: % of rated power
3.ReactiveCurrentReference	: ID1459, unit: % of rated power
4.FrequencyDroop			: ID1534, unit: Hz
5.VoltageDroop				: ID1535, unit: % of Nominal Voltage
6.FrequencyDroopOffset		: ID1791, unit: Hz
7.VoltageCorrection			: ID1790, unit: V
8.BaseRefRampRate			: ID1536, unit: % base current ref / s 
9.StartPowerMode			: ID1503, 0: Start zero activePower D7 card, 1: start zero activepower drive, 2: Droop, 3: Isochronous (keep reference)
10.StartVoltageMode			: ID1641, 0:Start zero reactive power D7 card, 1: Droop, 2: Keep Reference
11.OutputActivePowerLimit	: ID1288, unit: % of rated current
12.InputActivePowerLimit 	: ID1287, unit: % of rated current
13.							: SPARE
14.							: SPARE
15.							: SPARE	
16.							: SPARE



OPTIONALLY:
IF above Powerlimit is not working in ugrid mode:
CurrentLimitMin
CurrentLimitMax
IF HV ramp is not working in ugrid, add
BaseCurrentRefRampRate 	:ID1536



DESCRIPTION:
Als er geen communicatie tussen parallele power systemen is: Droop mode of start zero Q/P
Als er WEL communicatie tussen parallele power systemen is: Keep reference 

*)
END_METHOD

END_FUNCTION_BLOCK

// ---- POUs/Functions-FBs-Programs/_generalFunctions/fb_MovingAverage.TcPOU
FUNCTION_BLOCK fb_MovingAverage
VAR_INPUT
	IN 		: REAL;
	length	: UINT;
	enable 	: BOOL;
END_VAR
VAR_OUTPUT
	Q : REAL;
END_VAR
VAR
	r_Sumvalue		: REAL;
	ui_Index		: UINT; 
END_VAR

IF enable THEN
	r_Sumvalue := r_sumvalue + IN;
	ui_Index := ui_index +1;
	
	IF ui_index > length THEN
		r_Sumvalue := r_Sumvalue - Q * (ui_index - length +1);
		ui_index := length - 1; 
	END_IF
	
	Q := r_Sumvalue / MAX(1, ui_Index); 
ELSE
	Q := IN;
	r_Sumvalue := 0;
	ui_Index := 0;
END_IF

END_FUNCTION_BLOCK

// ---- POUs/Objects/PowerStack/PowerModule/FB_PowerModule_Buscoupler.TcPOU
FUNCTION_BLOCK FB_PowerModule_Buscoupler
VAR_IN_OUT
	get									: ST_PowerModule_Get;
	b_MccbEDM							: BOOL;
END_VAR

VAR_INPUT
	b_MCCBChargeSpring					: BOOL := TRUE;
	b_DCmainContactor					: BOOL := FALSE;
	b_DCprechargeContactor				: BOOL := FALSE;
	b_FanOn								: BOOL := FALSE;
	b_D7SyncRq							: BOOL := FALSE;
END_VAR

VAR
	a_StatusDataIN				AT %I* : ARRAY[1..1] OF UINT;
	a_EL2008					AT %Q* : ARRAY[1..8] OF BOOL;
	a_EL1008					AT %I* : ARRAY[1..8] OF BOOL;
	a_EL3208					AT %I* : ARRAY[1..8] OF ST_AnalogInputData;
	AdditionalMeasurements		: FB_Powermodule_additionalMeasurements;
END_VAR

b_MCCBChargeSpring := TRUE; // NOT get.b_MccbTripOK;

read();

Write();

AdditionalMeasurements(Get := get);

METHOD Read

VAR
	r_precision	: REAL := 0.1;
	i			: INT;
END_VAR

var_inst
	ton_FlowOK	:	Ton := (pt := T#5s);
END_VAR


//Mapping input data
get.ui_BuscouplerCommStatus				:= a_StatusDataIN[1];
 

// booleans can be written directly
get.b_MccbTripOK						:= a_EL1008[1];
b_MccbEDM								:= a_EL1008[2];
get.b_FanFb								:= a_EL1008[3];
get.b_MccbUvr24VdcOK					:= a_EL1008[4];
get.b_DCcontactorFb						:= a_EL1008[5];
ton_FlowOK(in							:= a_EL1008[6]);

get.b_FlowSwitchOK	 := ton_FlowOK.q;	
// scale temperature measurements
get.r_TemperatureCMChoke[1] := a_EL3208[1].Value * r_precision;
get.r_TemperatureCMChoke[2] := a_EL3208[2].Value * r_precision;
get.r_TemperatureCMChoke[3] := a_EL3208[3].Value * r_precision;
get.r_TemperatureCMChoke[4] := a_EL3208[4].Value * r_precision;
get.r_TemperatureGridchoke[1] := a_EL3208[5].Value * r_precision;
get.r_TemperatureGridchoke[2]  := a_EL3208[6].Value * r_precision;
get.r_TemperatureGridchoke[3]  := a_EL3208[7].Value * r_precision;
//spare := a_EL3208[8] * r_precision;

get.Events.b_PT100Underrange := FALSE;
get.Events.b_PT100Overrange := FALSE;
get.Events.by_PT100ErrorCount := 0;
FOR i := 1 TO 8 DO
	IF a_EL3208[i].Status.Underrange THEN get.Events.b_PT100Underrange := TRUE; END_IF;
	IF a_EL3208[i].Status.Overrange THEN get.Events.b_PT100Overrange := TRUE; END_IF;
	IF a_EL3208[i].Status.Error THEN get.Events.by_PT100ErrorCount := get.Events.by_PT100ErrorCount +1; END_IF;
END_FOR
END_METHOD

METHOD Write
(*NOTE: the input bit array of the el2008 has by default wrong naming. The hardware IO arrangement is from top to bottom columnswise.
While software linked IO is from left to right, row wise.
 The name cannot be changed. It is inconvenient to adjust the GSDML file as it comes from the internal libary.
This solved in the mapping between IO and a_EL2008 output array*)

a_EL2008[5]	:= b_DCprechargeContactor;
a_EL2008[4]	:= b_DCmainContactor;
a_EL2008[3] := TRUE;// b_MCCBChargeSpring; // MCCB reset
a_EL2008[2] := b_fanOn;
a_EL2008[1] := b_D7SyncRq;
END_METHOD

END_FUNCTION_BLOCK

// ---- POUs/Objects/PowerStack/PowerModule/FB_Powermodule_additionalMeasurements.TcPOU
FUNCTION_BLOCK FB_Powermodule_additionalMeasurements 
VAR_IN_OUT
	get									: ST_PowerModule_Get;
END_VAR


VAR
	a_EL3208_1					AT %I* : ARRAY[1..8] OF ST_AnalogInputData;
	a_EL3208_2					AT %I* : ARRAY[1..8] OF ST_AnalogInputData;
	a_EL3208_3					AT %I* : ARRAY[1..8] OF ST_AnalogInputData;
	a_EL3208_4					AT %I* : ARRAY[1..8] OF ST_AnalogInputData;
	r_precision	: REAL := 0.1;
	i : INT;
END_VAR

get.AddTemperatures.r_CMchokeInner[1] 		:= a_EL3208_1[1].value * r_precision; 
get.AddTemperatures.r_CMchokeInner[2] 		:= a_EL3208_1[2].value * r_precision; // L2
get.AddTemperatures.r_CMchokeInner[3] 		:= a_EL3208_1[3].value * r_precision; // l3
get.AddTemperatures.r_CMchokeInner[4] 		:= a_EL3208_1[4].value * r_precision; // DC
get.AddTemperatures.r_GrChokeInner[1] 		:= a_EL3208_1[5].value * r_precision; // L1
get.AddTemperatures.r_GrChokeInner[2] 		:= a_EL3208_1[6].value * r_precision; // L2
get.AddTemperatures.r_GrchokeInner[3] 		:= a_EL3208_1[7].value * r_precision; // L3
get.AddTemperatures.r_ambient 				:= a_EL3208_1[8].value * r_precision; //
get.AddTemperatures.r_CMchokeOuter[1] 		:= a_EL3208_2[1].value * r_precision; // L1
get.AddTemperatures.r_CMchokeOuter[2] 		:= a_EL3208_2[2].value * r_precision; // L2
get.AddTemperatures.r_CMchokeOuter[3] 		:= a_EL3208_2[3].value * r_precision; // L3
get.AddTemperatures.r_CMchokeOuter[4] 		:= a_EL3208_2[4].value * r_precision; // DC
get.AddTemperatures.r_GrChokeOuter[1] 		:= a_EL3208_2[5].value * r_precision;	//
get.AddTemperatures.r_GrChokeOuter[2] 		:= a_EL3208_2[6].value * r_precision; //
get.AddTemperatures.r_GrChokeOuter[3] 		:= a_EL3208_2[7].value * r_precision; // L3
get.AddTemperatures.r_FancoilCompartement 	:= a_EL3208_2[8].value * r_precision; //
get.AddTemperatures.r_ACCapsBottom 			:= a_EL3208_3[1].value * r_precision; // 
get.AddTemperatures.r_AcCapsTop			 	:= a_EL3208_3[2].value * r_precision; //
get.AddTemperatures.r_DcCaps			 	:= a_EL3208_3[3].value * r_precision; // 
get.AddTemperatures.r_ACbusbarOutput		:= a_EL3208_3[4].value * r_precision; //
get.AddTemperatures.r_ACbusbarCMChoke 		:= a_EL3208_3[5].value * r_precision; // 
get.AddTemperatures.r_DCbusbarCMChoke 		:= a_EL3208_3[6].value * r_precision; // 
get.AddTemperatures.r_WaterInletFancoil		:= a_EL3208_4[1].value * r_precision; //
get.AddTemperatures.r_AirOutletFancoil 		:= a_EL3208_4[2].value * r_precision; //
get.AddTemperatures.r_WaterOutletFancoil	:= a_EL3208_4[3].value * r_precision; //
get.AddTemperatures.r_AirInletModule		:= a_EL3208_4[4].value * r_precision; //

FOR i := 1 TO 8 DO
	IF a_EL3208_1[i].Status.Underrange THEN get.Events.b_PT100Underrange := TRUE; END_IF;
	IF a_EL3208_1[i].Status.Overrange THEN get.Events.b_PT100Overrange := TRUE; END_IF;
	IF a_EL3208_1[i].Status.Error THEN get.Events.by_PT100ErrorCount := get.Events.by_PT100ErrorCount +1; END_IF;
	IF a_EL3208_2[i].Status.Underrange THEN get.Events.b_PT100Underrange := TRUE; END_IF;
	IF a_EL3208_2[i].Status.Overrange THEN get.Events.b_PT100Overrange := TRUE; END_IF;
	IF a_EL3208_2[i].Status.Error THEN get.Events.by_PT100ErrorCount := get.Events.by_PT100ErrorCount +1; END_IF;
END_FOR
FOR i := 1 TO 6 DO
	IF a_EL3208_3[i].Status.Underrange THEN get.Events.b_PT100Underrange := TRUE; END_IF;
	IF a_EL3208_3[i].Status.Overrange THEN get.Events.b_PT100Overrange := TRUE; END_IF;
	IF a_EL3208_3[i].Status.Error THEN get.Events.by_PT100ErrorCount := get.Events.by_PT100ErrorCount +1; END_IF;
END_FOR
FOR i := 1 TO 4 DO
	IF a_EL3208_4[i].Status.Underrange THEN get.Events.b_PT100Underrange := TRUE; END_IF;
	IF a_EL3208_4[i].Status.Overrange THEN get.Events.b_PT100Overrange := TRUE; END_IF;
	IF a_EL3208_4[i].Status.Error THEN get.Events.by_PT100ErrorCount := get.Events.by_PT100ErrorCount +1; END_IF;
END_FOR

END_FUNCTION_BLOCK

// ---- POUs/Functions-FBs-Programs/fb_Ramp_dual.TcPOU
FUNCTION_BLOCK fb_Ramp_dual
VAR_INPUT
	SetZero		: BOOL;
	SetToIN		: BOOL;
	IN			: REAL;
	rampDown	: REAL;
	RampUp	: REAL;
	Enable	: BOOL;
END_VAR
VAR_OUTPUT
	Q		: REAL;
END_VAR

VAR
	r_RampFinal				: REAL;
	fb_ramp					: FB_CTRL_RAMP_GENERATOR;
	st_ParamsRamp    		: ST_CTRL_RAMP_GENERATOR_PARAMS;
	r_inLast				: REAL;
END_VAR

IF SetZero THEN
	IN := 0;
END_IF

IF SETtoIN OR SetZero THEN
	RampUp := 10000;
	rampDown := 100000;
END_IF

st_ParamsRamp.fVeloNeg := rampDown;
st_ParamsRamp.fVeloPos := RampUp;
st_ParamsRamp.tCtrlCycleTime := T#1MS;
st_ParamsRamp.tTaskCycleTime := T#1MS;
fb_ramp(
	bEnable:= Enable,
	fout => Q,
	stParams := st_ParamsRamp,
	fStart:= r_inlast,
	fTarget:= IN);
	

IF fb_ramp.bValueReached AND Enable THEN
	r_inlast := IN;
END_IF

IF NOT Enable THEN
	Q := IN;
END_IF

END_FUNCTION_BLOCK

// ---- POUs/Functions-FBs-Programs/_acFunctions/fb_LOMdetection.TcPOU
FUNCTION_BLOCK fb_LOMdetection
VAR_INPUT
	r_Freq		: REAL;
	r_NomFreq	: REAL;
	r_volt		: REAL;
	b_enable	: BOOL;
	SlowDetection	: BOOL;
END_VAR
VAR_IN_OUT CONSTANT
	st_params : ST_Powerstack_LOMparams;
END_VAR

VAR_OUTPUT
	Q	: BOOL;
END_VAR
VAR	
	nomFreq					:  REAL;
	tofQTripTime		: TOF := (PT := T#1S);
	ton_Reset : TON 		:= (PT := T#1S);
	ton_FreqNOKDelay1		: TON := (PT := T#2S);
	ton_FreqNOKDelay2		: TON := (PT := T#0.2S);
	FreqThreshold1			: REAL := 0.2;
	ton_VoltNOKDelay		: TON := (PT := T#2S);
	FreqMin					: REAL;
	FreqMax					: REAL;
	b_FreqNOK			: BOOL;
END_VAR

Nomfreq := settings.GridParams.r_GridNominalFrequency;
FreqMin	:= settings.GridParams.r_GridFrequencyMin;
FreqMax	:= settings.GridParams.r_GridFrequencyMax;
ton_FreqNOKDelay1(IN := LIMIT(Nomfreq - FreqThreshold1, r_Freq, Nomfreq + FreqThreshold1) <> r_freq,
	PT := SEL(SlowDetection, T#0.5S, T#3S)
		);
ton_FreqNOKDelay2(IN := LIMIT(FreqMin, r_Freq, FreqMax) <> r_freq);
ton_VoltNOKDelay(IN := NOT ACvoltageCheck(IN := r_Volt));
tofQTripTime(Q => Q);

tofQTripTime.IN := (rocof(
	frequency :=  r_freq, 
	NomFrequency := r_nomFreq,)
	OR
	ton_FreqNOKDelay1.Q
	OR
	ton_FreqNOKDelay2.Q 
	OR
	ton_VoltNOKDelay.Q)
	AND
	b_enable;
	
ton_Reset();

METHOD Reset : BOOL
VAR_INPUT
END_VAR

VAR_INST
	
END_VAR
ton_Reset.IN := Q;

IF NOT Q THEN
	ton_Reset.IN := FALSE;
	Reset := TRUE;
END_IF
END_METHOD

METHOD RoCoF : BOOL
VAR_INPUT
	frequency	: REAL;
	NomFrequency: REAL;
END_VAR

VAR_INST
	FastmodeDelay	: TON := (PT := T#2s);
	t_detectionTime	: TIME;
	FrequencyMA		: FB_movingaverage := (enable := TRUE);
	rocofLast		: REAL;
	FreqLast		: REAL;
	FreqDelta		: REAL;	
	DetectionTimer	: TON;
	RoCofAct		: REAL;
	LomDetected		: BOOL;
END_VAR
FrequencyMA(IN := Frequency, length :=  st_params.FreqFilterLength);

FastModeDelay(IN := NOT SlowDetection AND NOT st_params.ForceSlowDetection);
t_DetectionTime := TO_TIME(SEL(FastModeDelay.Q, st_params.DetectionTimeSlow_ms, st_params.DetectionTimeFast_ms));
detectionTimer(IN := NOT detectiontimer.Q, PT := t_DetectionTime );

IF detectionTimer.Q THEN
	RocofAct := (FrequencyMA.Q - FreqLast) / (MAX(1, TO_REAL(t_DetectionTime)) * 0.001);
	FreqLast:= FrequencyMA.Q;
END_IF

IF ABS(rocofLast) < ABS(rocofAct) THEN
	rocofLast := rocofAct;
END_IF

IF ABS(RocofAct) > st_params.RoCoFlimit * SEL(SlowDetection, 1, 4) AND b_Enable THEN
	LomDetected := TRUE;
END_IF

IF ton_Reset.Q OR NOT b_enable THEN
	rocofLast := 0;
	LomDetected := FALSE;
END_IF

Rocof := LomDetected;
END_METHOD

END_FUNCTION_BLOCK

// ---- POUs/Functions-FBs-Programs/_generalFunctions/Between.TcPOU
FUNCTION Between : BOOL
VAR_INPUT
	in			: REAL;
	lim1		: REAL;
	lim2		: REAL;
END_VAR
VAR
END_VAR

IF lim1 > lim2 THEN 
		IF (in <= lim1) AND (in >= lim2) THEN
			Between:=TRUE;
		ELSE
			Between:=FALSE;
		END_IF

ELSE
		IF (in >= lim1) AND (in <= lim2) THEN
			Between:=TRUE;
		ELSE
			Between:=FALSE;
		END_IF	
END_IF

END_FUNCTION

// ---- POUs/Objects/PowerQualityMonitor/FB_PowerQualityMonitoring.TcPOU
FUNCTION_BLOCK FB_PowerQualityMonitoring
VAR PERSISTENT
	r_BESSEnergySupplied		: REAL;
	r_BESSEnergyConsumed		: REAL;
END_VAR


VAR_OUTPUT
	get							: ST_PowerMonitor_get;
END_VAR

VAR_INPUT
	b_Enable					: 	BOOL;
	PowerStackGet				:	st_Powerstack_Get;
	b_TNModeActive				:	BOOL;
	b_ThirdOutputFieldAvailable	: 	BOOL;
	b_InputFieldsAvailable		: 	BOOL;
	b_NeutralTransformerAvailable: BOOL;
END_VAR

VAR
	EL3453_Input	: FB_EL3453;
	EL3453_Output	: FB_EL3453;
END_VAR

//INSTANCIATE FBS
EL3453_Input();
EL3453_Output();


MapPowerstackGetToGetStruct();

CalcBessEnergyValues(P := get.inverter.ar_ActivePower[0], ESupplied => get.Inverter.r_EnergySupplied, EConsumed => get.Inverter.r_EnergyConsumed);

GetLoadshares(powerstackGet.r_RatedPower, get.InputField.ar_ApparentPower[0], get.OutputField.ar_ApparentPower[0]);

METHOD CalcBessEnergyValues

VAR_INPUT
	P	: REAL; //active power
END_VAR

VAR_INST
	ton_CumEnergy		: TON := (PT:= T#1MS);
END_VAR

VAR_OUTPUT
	Esupplied	: REAL;
	EConsumed 	: REAL;
END_VAR
ton_CumEnergy(IN:= NOT ton_CumEnergy.Q);

IF ton_CumEnergy.Q THEN
	IF P > 0 THEN
		r_BESSEnergySupplied := r_BESSEnergySupplied + ABS(P) / 3600000;
	ELSIF P < 0 THEN
		r_BESSEnergyConsumed := r_BESSEnergyConsumed + ABS(P) / 3600000;
	END_IF	
END_IF


//Set persistent values to get struct.
Esupplied := r_BESSEnergySupplied;
EConsumed := r_BESSEnergyConsumed;
END_METHOD

METHOD PUBLIC EMstop : BOOL
//returns true when ready/stopped
END_METHOD

METHOD GetDiagnostics
VAR_IN_OUT
	AddError		: ARRAY [*] OF FB_AddErrorST;
	a_ActiveEvents	: ARRAY [*] OF ST_ErrorStruct;
	w_Index			: WORD;
END_VAR
//JANITZA
(*Comm Warning*)		AddError[w_Index](
		b_ErrorTrig			:= get.events.b_MBCommWarning,
		out_ST_Error			:= a_ActiveEvents[w_Index],
		w_ErrorID					:= 1,
		e_ObjectID				:= eObject_ID.PowerMonitor,
		s_Message				:= 'janitza communication warning',
		e_sev					:= eseverity.warning
	);
	w_Index := w_Index +1;
	
(*Comm timeout*)		AddError[w_Index](
		b_ErrorTrig			:= get.events.b_MBTimeoutWarning,
		out_ST_Error			:= a_ActiveEvents[w_Index],
		w_ErrorID					:= 2,
		s_Message				:= 'janitza communication timeout',
		e_sev					:= eseverity.Warning
	);
	w_Index := w_Index +1;
	
(*Comm fault*)		AddError[w_Index](
		b_ErrorTrig			:= get.events.b_MBCommError,
		out_ST_Error			:= a_ActiveEvents[w_Index],
		w_ErrorID					:= 3,
		t_TriggerTime		:= T#10S,
		s_Message				:= 'janitza communication fault',
		e_sev					:= eseverity.Normalshutdown
	);
	w_Index := w_Index +1;
	
//EL3443
(*Comm Warning*)		AddError[w_Index](
		b_ErrorTrig			:= get.events.b_EL3443Warning,
		out_ST_Error			:= a_ActiveEvents[w_Index],
		w_ErrorID					:= 4,
		s_Message				:= 'EL3443 powermonitor warning',
		e_sev					:= eseverity.Warning,
	);
	w_Index := w_Index +1;
END_METHOD

METHOD GetLoadshares : BOOL
VAR_INPUT
	r_ratedPower		: REAL;
	r_InputPower		: REAL;
	r_OutputPower		: REAL;
END_VAR
get.InputField.r_loadshare := r_InputPower / MAX(1, r_ratedPower) * 100;
get.OutputField.r_loadshare := r_OutputPower / MAX(1, r_ratedPower) * 100;
END_METHOD

METHOD MapInputPmsToGetStruct : BOOL
VAR_INPUT
END_VAR
END_METHOD

METHOD MapOutputPmsToGetStruct : BOOL
VAR_INPUT
END_VAR
END_METHOD

METHOD MapPowerstackGetToGetStruct
//Voltage dependent values of Internal supply are copied from outputfield, but are only valid if netcontactor is closed.
IF powerstackget.Netcontactor.b_NetConFb THEN
	get.inverter.ar_LineVoltage[0] := powerstackGet.r_ACVoltageD7;
	get.inverter.ar_Frequency[0] := powerstackGet.r_FrequencyD7;
ELSE
	get.inverter.ar_LineVoltage[0] := powerstackGet.r_ACVoltageSupply;
	get.inverter.ar_Frequency[0] := powerstackGet.r_FrequencySupply;
END_IF

//Fill BESS data with PowerStackData
//Not all data is filled in here, determine which are desired and possible.
get.inverter.e_ACrotationStatus := get.OutputField.e_ACrotationStatus;
//phase currents not available at this time, only the average is set
get.inverter.ar_Current[0] := PowerStackGet.r_AcCurrent;

//phase Powers not available at this time, only the average is set
Get.inverter.ar_ApparentPower[0]	:=	PowerStackGet.r_ApparentPower;
Get.inverter.ar_ReactivePower[0]	:=	PowerStackGet.r_ReactivePower;
Get.inverter.ar_ActivePower[0]		:=	PowerStackGet.r_ActivePower;


//phase Powerfactors not available at this time, only the average is set									
Get.inverter.ar_PowerFactor[0]		:=	PowerStackGet.r_CosPhi;
END_METHOD

METHOD Public Reset : BOOL
//clear data struct
//reinitialize janitza + el3443
//clear all errors?

//returns true when ready
Reset := NOT get.events.b_MBCommError;
END_METHOD

END_FUNCTION_BLOCK

// ---- POUs/Functions-FBs-Programs/IO_modules/Beckhoff/FB_EL3453.TcPOU
FUNCTION_BLOCK FB_EL3453

VAR_OUTPUT	
	Diagnostics					: MDP5001_341_I_C314AD31;
	General						: ST_PQVoltageData;
	Status						: ST_PQstatusData;
	Quality						: ST_PQGridQualityData;	
	ConfiguredCtRatio			: ARRAY [1..4] OF REAL;		
END_VAR

VAR
	EL3453 						: MDP5001_341_6E3B8FF1;
	DiagData					: MDP5001_341_C314AD31;
		
	VRatio  				: REAL := 1;
	CRatio  				: REAL := 1000;
	CInverse				: BOOL := FALSE; 
	
	
	bInitDone				: BOOL;
END_VAR

Diagnostics := DiagData.MDP5001_341_Input;
General:= PQVoltageData();
Quality := GridQuality();
Status:= Status;

GetPMXsettings(b_start := NOT bInitDone);

bInitDone := TRUE;

METHOD DynamicRatio
VAR_INPUT
	VPrimair  				: REAL := 400;
	VSecundair				: REAL := 400;
	CtRatio  				: UINT := 1000;
	CTInverse				: BOOL := FALSE; 
END_VAR

VAR_INST	
	OverCurrentThreshold : REAL := 1.05;
	FrequencyOkLowLimit : REAL := 45;
	FrequencyOkHighLimit : REAL := 65;
	VoltageOkHighLimitPU : REAL := 1.1;
	VoltageOkLowLimitPU : REAL := 0;
END_VAR

VAR
	i : INT;
	PhaseError :BOOL;
END_VAR

VAR_OUTPUT
	Status					 : ST_PQstatusData;
	b_VoltagesOK			 : BOOL;
	e_ACrotationState		 : eACRotationState;
	ar_PhaseVoltage			 : ARRAY [0..3] OF REAL;
	ar_LineVoltage			 : ARRAY [0..3] OF REAL;
	ar_Current				 : ARRAY [0..4] OF REAL;
	ar_ActivePower			 : ARRAY [0..3] OF REAL;
	ar_ReactivePower		 : ARRAY [0..3] OF REAL;
	ar_ApparentPower		 : ARRAY [0..3] OF REAL;
	ar_PowerFactor			 : ARRAY [0..3] OF REAL;
	ar_Frequency			 : ARRAY [0..3] OF REAL;
	r_voltageUnbalance		 : REAL;
	r_CurrentUnbalance		 : REAL;
END_VAR

VAR
	ReactiveDirection			: SINT;
END_VAR
IF VPrimair = 0 OR VSecundair = 0 THEN
	Status.b_SettingFault := TRUE;
	RETURN;
END_IF

VRatio := Vprimair / Vsecundair;
CRatio := CtRatio;
CInverse := CTInverse;

//current
ar_Current[1]:= ValueConversion(DataSelector._C, ABS(EL3453.MDP5001_341_Input.L1_Classic_Current));
ar_Current[2]:= ValueConversion(DataSelector._C, ABS(EL3453.MDP5001_341_Input.L2_Classic_Current));
ar_Current[3]:= ValueConversion(DataSelector._C, ABS(EL3453.MDP5001_341_Input.L3_Classic_Current));
ar_Current[0] := (ar_Current[1] + ar_Current[2] + ar_Current[3]) / 3;

//voltage
ar_PhaseVoltage[1] := ValueConversion(DataSelector._V, EL3453.MDP5001_341_Input.L1_Classic_Voltage);
ar_PhaseVoltage[2] := ValueConversion(DataSelector._V, EL3453.MDP5001_341_Input.L2_Classic_Voltage);
ar_PhaseVoltage[3] := ValueConversion(DataSelector._V, EL3453.MDP5001_341_Input.L3_Classic_Voltage);
ar_PhaseVoltage[0] := (ar_PhaseVoltage[1] + ar_PhaseVoltage[2] + ar_PhaseVoltage[3]) / 3;

ar_LineVoltage[1]:= ar_PhaseVoltage[1]* 1.73;
ar_LineVoltage[2]:= ar_PhaseVoltage[2]* 1.73;
ar_LineVoltage[3]:= ar_PhaseVoltage[3]* 1.73;
ar_LineVoltage[0] := ar_PhaseVoltage[0] * 1.73;

IF VRatio <> 0 THEN
	b_VoltagesOK:= ACPhasesOK(ar_LineVoltage[1] / VRatio, ar_LineVoltage[2] / VRatio, ar_LineVoltage[3] / VRatio);
END_IF
e_ACrotationState	:= GetRotatingField(EL3453.MDP5001_341_Input.Total_Status_Grid_Direction, b_VoltagesOk);


//active power
ar_ActivePower[1]:= ValueConversion(DataSelector._P, EL3453.MDP5001_341_Input.L1_Classic_Active_power);
ar_ActivePower[2]:= ValueConversion(DataSelector._P, EL3453.MDP5001_341_Input.L2_Classic_Active_power);
ar_ActivePower[3]:= ValueConversion(DataSelector._P, EL3453.MDP5001_341_Input.L3_Classic_Active_power);
ar_ActivePower[0] := (ar_ActivePower[1] + ar_ActivePower[2] + ar_ActivePower[3]);

//Reactive power
IF EL3453.MDP5001_341_Input.Total_Reactive_Fundamental_Reactive_Power_Fund < 0 THEN ReactiveDirection := -1; ELSE ReactiveDirection := 1; END_IF
ar_ReactivePower[1]:= ReactiveDirection * ValueConversion(DataSelector._Q, EL3453.MDP5001_341_Input.L1_Classic_Reactive_power);
ar_ReactivePower[2]:= ReactiveDirection * ValueConversion(DataSelector._Q, EL3453.MDP5001_341_Input.L2_Classic_Reactive_power);
ar_ReactivePower[3]:= ReactiveDirection * ValueConversion(DataSelector._Q, EL3453.MDP5001_341_Input.L3_Classic_Reactive_power);
ar_ReactivePower[0] := (ar_ReactivePower[1] + ar_ReactivePower[2] + ar_ReactivePower[3]);

//Apparent power
ar_ApparentPower[1]:= ValueConversion(DataSelector._S, EL3453.MDP5001_341_Input.L1_Classic_Apparent_power);
ar_ApparentPower[2]:= ValueConversion(DataSelector._S, EL3453.MDP5001_341_Input.L2_Classic_Apparent_power);
ar_ApparentPower[3]:= ValueConversion(DataSelector._S, EL3453.MDP5001_341_Input.L3_Classic_Apparent_power);
ar_ApparentPower[0] := (ar_ApparentPower[1] + ar_ApparentPower[2] + ar_ApparentPower[3]);

//Frequecny
ar_Frequency[1] := ValueConversion(DataSelector._F, EL3453.MDP5001_341_Input.L1_Classic_Frequency);
ar_Frequency[2] := ValueConversion(DataSelector._F, EL3453.MDP5001_341_Input.L2_Classic_Frequency);
ar_Frequency[3] := ValueConversion(DataSelector._F, EL3453.MDP5001_341_Input.L3_Classic_Frequency);
ar_Frequency[0]	:= (ar_Frequency[1] + ar_Frequency[2] + ar_Frequency[3]) / 3;

ar_PowerFactor [1] := Powerfactor(ar_ActivePower[1], ar_ApparentPower[1], ar_ReactivePower[1]);
ar_PowerFactor [2] := Powerfactor(ar_ActivePower[2], ar_ApparentPower[2], ar_ReactivePower[2]);
ar_PowerFactor [3] := Powerfactor(ar_ActivePower[3], ar_ApparentPower[3], ar_ReactivePower[3]);
ar_PowerFactor [0] := Powerfactor(ar_ActivePower[0], ar_ApparentPower[0], ar_ReactivePower[0]);
r_VoltageUnbalance := LineUnbalance(ar_LineVoltage[1], ar_LineVoltage[2], ar_LineVoltage[3]);
r_CurrentUnbalance := LineUnbalance(ar_Current[1], ar_Current[2], ar_Current[3]);

//loop through phases 
FOR i := 1 TO 3 DO
	PhaseError := FALSE;
	
	IF ar_Current[i] >= OverCurrentThreshold * CtRatio THEN
		Status.b_OverCurrent := TRUE;
		PhaseError := TRUE;
	END_IF
	
	IF LIMIT(VoltageOKLowLimitPU * Vsecundair, ar_LineVoltage[i], VoltageOKHighLimitPU * VSecundair) <> ar_LineVoltage[i] THEN
		Status.b_OverVoltage := ar_lineVoltage[i] >= VoltageOKHighLimitPU * VSecundair;
		Status.b_UnderVoltage := ar_lineVoltage[i] <= VoltageOKLowLimitPU * VSecundair;
		PhaseError := TRUE;
	END_IF
	
	IF LIMIT(FrequencyOKLowLimit, ar_Frequency[i], FrequencyOKHighLimit) <> ar_Frequency[i] THEN
		PhaseError := TRUE;
		status.b_OverFrequency := ar_Frequency[i] >= FrequencyOKHighLimit;
		status.b_UnderFrequency := ar_Frequency[i] <= FrequencyOKLowLimit;
	END_IF
	
	IF phaseError THEN
		status.b_Fault := TRUE;
		status.b_Error_Phase[i] := PhaseError;
	END_IF
END_FOR
END_METHOD

//FB_Init is always available implicitly and it is used primarily for initialization.
//The return value is not evaluated. For a specific influence, you can also declare the
//methods explicitly and provide additional code there with the standard initialization
//code. You can evaluate the return value.
METHOD FB_Init: BOOL
VAR_INPUT
    bInitRetains: BOOL; // TRUE: the retain variables are initialized (reset warm / reset cold)
    bInCopyCode: BOOL;  // TRUE: the instance will be copied to the copy code afterward (online change)   
END_VAR
bInitDone := FALSE;
END_METHOD

METHOD FixedRatio: BOOL
VAR_INPUT
END_VAR

VAR_INST
	b_VoltagesOk : BOOL;
END_VAR

VAR_OUTPUT
	Status 			: ST_PQStatusData;
	Measurements 	: ST_PQVoltageData;
END_VAR
//General stuff
b_VoltagesOk							:= ACphasesOK(EL3453.MDP5001_341_Input.Total_L_L_Voltages_L1_L2_Voltage, EL3453.MDP5001_341_Input.Total_L_L_Voltages_L2_L3_Voltage, EL3453.MDP5001_341_Input.Total_L_L_Voltages_L3_L1_Voltage);
Measurements.b_VoltagesOK				:= b_VoltagesOk;
Measurements.e_ACrotationStatus			:= GetRotatingField(EL3453.MDP5001_341_Input.Total_Status_Grid_Direction, b_VoltagesOk);
Measurements.ar_phaseVoltage[1]			:= EL3453.MDP5001_341_Input.L1_Basic_Voltage;
Measurements.ar_phaseVoltage[2]			:= EL3453.MDP5001_341_Input.L2_Basic_Voltage;
Measurements.ar_phaseVoltage[3]			:= EL3453.MDP5001_341_Input.L3_Basic_Voltage;
Measurements.ar_PhaseVoltage[0] 			:= (EL3453.MDP5001_341_Input.L1_Basic_Voltage + EL3453.MDP5001_341_Input.L2_Basic_Voltage + EL3453.MDP5001_341_Input.L3_Basic_Voltage) / 3;
Measurements.ar_LineVoltage[1] 			:= EL3453.MDP5001_341_Input.Total_L_L_Voltages_L1_L2_Voltage;
Measurements.ar_LineVoltage[2] 			:= EL3453.MDP5001_341_Input.Total_L_L_Voltages_L2_L3_Voltage;
Measurements.ar_LineVoltage[3] 			:= EL3453.MDP5001_341_Input.Total_L_L_Voltages_L3_L1_Voltage;
Measurements.ar_LineVoltage[0] 			:= (EL3453.MDP5001_341_Input.Total_L_L_Voltages_L1_L2_Voltage + EL3453.MDP5001_341_Input.Total_L_L_Voltages_L2_L3_Voltage + EL3453.MDP5001_341_Input.Total_L_L_Voltages_L3_L1_Voltage) / 3;
Measurements.ar_PowerFactor[1] 			:= EL3453.MDP5001_341_Input.L1_Power_Power_Factor;
Measurements.ar_PowerFactor[2] 			:= EL3453.MDP5001_341_Input.L2_Power_Power_Factor;
Measurements.ar_PowerFactor[3] 			:= EL3453.MDP5001_341_Input.L3_Power_Power_Factor;
Measurements.ar_PowerFactor[0] 			:= EL3453.MDP5001_341_Input.Total_Basic_Power_Factor;
Measurements.ar_current[1]					:= EL3453.MDP5001_341_Input.L1_Basic_Current;
Measurements.ar_current[2]					:= EL3453.MDP5001_341_Input.L2_Basic_Current;
Measurements.ar_current[3]					:= EL3453.MDP5001_341_Input.L3_Basic_Current;
Measurements.ar_current[4]					:= EL3453.MDP5001_341_Input.Total_Basic_Neutral_Line_Current;
Measurements.ar_Current[0]					:= (EL3453.MDP5001_341_Input.L1_Basic_Current + EL3453.MDP5001_341_Input.L2_Basic_Current + EL3453.MDP5001_341_Input.L3_Basic_Current) / 3;
Measurements.ar_activePower[1]				:= EL3453.MDP5001_341_Input.L1_Power_Fundamental_active_Power_Fund;
Measurements.ar_activePower[2]				:= EL3453.MDP5001_341_Input.L2_Power_Fundamental_active_Power_Fund;
Measurements.ar_activePower[3]				:= EL3453.MDP5001_341_Input.L3_Power_Fundamental_active_Power_Fund;
Measurements.ar_activePower[0]				:= EL3453.MDP5001_341_Input.Total_active_Fundamental_active_Power_Fund;
Measurements.ar_ReactivePower[1]			:= EL3453.MDP5001_341_Input.L1_Power_Fundamental_Reactive_Power_Fund;
Measurements.ar_ReactivePower[2]			:= EL3453.MDP5001_341_Input.L2_Power_Fundamental_Reactive_Power_Fund;
Measurements.ar_ReactivePower[3]			:= EL3453.MDP5001_341_Input.L3_Power_Fundamental_Reactive_Power_Fund;
Measurements.ar_ReactivePower[0]			:= EL3453.MDP5001_341_Input.Total_Reactive_Fundamental_Reactive_Power_Fund;
Measurements.ar_ApparentPower[1]			:= EL3453.MDP5001_341_Input.L1_Power_Apparent_Power;
Measurements.ar_ApparentPower[2]			:= EL3453.MDP5001_341_Input.L2_Power_Apparent_Power;
Measurements.ar_ApparentPower[3]			:= EL3453.MDP5001_341_Input.L3_Power_Apparent_Power;
Measurements.ar_ApparentPower[0]			:= EL3453.MDP5001_341_Input.Total_Apparent_Apparent_Power;
Measurements.r_VoltageUnbalance			:= EL3453.MDP5001_341_Input.Total_Advanced_Voltage_Unbalance;
Measurements.r_CurrentUnbalance			:= LineUnbalance(EL3453.MDP5001_341_Input.L1_Basic_Current, EL3453.MDP5001_341_Input.L2_Basic_Current, EL3453.MDP5001_341_Input.L3_Basic_Current);
Measurements.ar_CurrentTHD[1]				:= EL3453.MDP5001_341_Input.L1_Advanced_Current_Total_Harmonic_Distortion;
Measurements.ar_CurrentTHD[2]				:= EL3453.MDP5001_341_Input.L2_Advanced_Current_Total_Harmonic_Distortion;
Measurements.ar_CurrentTHD[3]				:= EL3453.MDP5001_341_Input.L3_Advanced_Current_Total_Harmonic_Distortion;
Measurements.ar_CurrentTHD[0]				:= EL3453.MDP5001_341_Input.Total_Advanced_Max_Current_Harmonic_Distortion;
Measurements.ar_VoltageTHD[1]				:= EL3453.MDP5001_341_Input.L1_Advanced_Voltage_Total_Harmonic_Distortion;
Measurements.ar_VoltageTHD[2]				:= EL3453.MDP5001_341_Input.L2_Advanced_Voltage_Total_Harmonic_Distortion;
Measurements.ar_VoltageTHD[3]				:= EL3453.MDP5001_341_Input.L3_Advanced_Voltage_Total_Harmonic_Distortion;
Measurements.ar_VoltageTHD[0]				:= EL3453.MDP5001_341_Input.Total_Advanced_Max_Voltage_Harmonic_Distortion;
Measurements.ar_Frequency[1] 				:= ValueConversion(DataSelector._F, EL3453.MDP5001_341_Input.L1_Classic_Frequency);
Measurements.ar_Frequency[2] 				:= ValueConversion(DataSelector._F, EL3453.MDP5001_341_Input.L2_Classic_Frequency);
Measurements.ar_Frequency[3] 				:= ValueConversion(DataSelector._F, EL3453.MDP5001_341_Input.L3_Classic_Frequency);
Measurements.ar_Frequency[0]				:= EL3453.MDP5001_341_Input.Total_Basic_Frequency;
Measurements.r_EnergyConsumed				:= TO_REAL(EL3453.MDP5001_341_Input.Total_Active_Active_Negative_Energy)/1000;
Measurements.r_EnergySupplied				:= TO_REAL(EL3453.MDP5001_341_Input.Total_Active_Active_Positive_Energy)/1000;
END_METHOD

METHOD GetPMXsettings
VAR_INPUT
	b_start : BOOL := TRUE;
END_VAR
 

VAR_INST
	PMXsettingsIndex			: ARRAY [1..4] OF WORD := [16#8000, 16#8100, 16#8200, 16#8300];
	SettingIndex				: BYTE := 16#12; //11 = voltage ratio, 12 = current ration
	fbReadCardParams			: FB_EcCoESdoRead;
	ratio						: FLOAT;
END_VAR
VAR
	i : INT;
	SnetID : STRING(23);
	AmsnetID : T_AmsNetID;
END_VAR
IF b_Start THEN
    fbReadCardParams(
        sNetID     := Tc2_System.F_CreateAmsNetId(DiagData.MDP5001_341_Input.AdsAddr.netId),
        nSlaveAddr := DiagData.MDP5001_341_Input.AdsAddr.port,
        nIndex     := PMXsettingsIndex[i],
        nSubIndex  := SettingIndex,
        pDstBuf    := ADR(ratio),
        cbBufLen   := SIZEOF(ratio),
        bExecute   := TRUE,
        tTimeOut   := T#2S,
    );

   IF NOT fbReadCardParams.bBusy AND fbReadCardParams.cbRead > 0 THEN
		IF NOT fbReadCardParams.bError THEN
			ConfiguredCtRatio[i] := ratio;
			i := i + 1;
		END_IF
   END_IF
END_IF
END_METHOD

METHOD PRIVATE GetRotatingField : eAcRotationState
VAR_INPUT
	b_Griddirection : BOOL;
	b_ACok			: BOOL;
END_VAR
IF NOT b_ACok THEN
	GetRotatingField := eAcRotationstate.None;
ELSE
	IF b_GridDirection = 1 THEN
		GetRotatingField := eAcRotationstate.Right;
	ELSE
		GetRotatingField := eAcRotationstate.Left;
	END_IF	
END_IF
END_METHOD

METHOD PRIVATE GridQuality : ST_PQGridQualityData;
IF EL3453.MDP5001_341_Input.L1_Status_Voltage_Sign_Bit THEN
	GridQuality.uli_TimeVoltZeroCrossup := EL3453.MDP5001_341_Input.L1_Timing_Voltage_Last_Zero_Crossing;
END_IF

GridQuality.b_SystemState 				:= EL3453.MDP5001_341_Input.Total_Status_System_State;
GridQuality.r_PowerQualityFactor 		:= EL3453.MDP5001_341_Input.Total_Status_Power_Quality_Factor;
GridQuality.r_Rocof 					:= EL3453.MDP5001_341_Input.Total_Basic_ROCOF;
END_METHOD

METHOD PRIVATE PQVoltageData : ST_PQVoltageData;

VAR_INST
	b_VoltagesOK 	: BOOL;
END_VAR
//General stuff
b_VoltagesOk								:= ACphasesOK(PQVoltageData.ar_LineVoltage[1], PQVoltageData.ar_LineVoltage[2], PQVoltageData.ar_LineVoltage[3]);
PQVoltageData.b_VoltagesOK					:= b_VoltagesOk;
PQVoltageData.e_ACrotationStatus			:= GetRotatingField(EL3453.MDP5001_341_Input.Total_Status_Grid_Direction, b_VoltagesOk);
PQVoltageData.ar_phaseVoltage[1]			:= EL3453.MDP5001_341_Input.L1_Basic_Voltage;
PQVoltageData.ar_phaseVoltage[2]			:= EL3453.MDP5001_341_Input.L2_Basic_Voltage;
PQVoltageData.ar_phaseVoltage[3]			:= EL3453.MDP5001_341_Input.L3_Basic_Voltage;
PQVoltageData.ar_PhaseVoltage[0] 			:= (EL3453.MDP5001_341_Input.L1_Basic_Voltage + EL3453.MDP5001_341_Input.L2_Basic_Voltage + EL3453.MDP5001_341_Input.L3_Basic_Voltage) / 3;
PQVoltageData.ar_LineVoltage[1] 			:= EL3453.MDP5001_341_Input.Total_L_L_Voltages_L1_L2_Voltage;
PQVoltageData.ar_LineVoltage[2] 			:= EL3453.MDP5001_341_Input.Total_L_L_Voltages_L2_L3_Voltage;
PQVoltageData.ar_LineVoltage[3] 			:= EL3453.MDP5001_341_Input.Total_L_L_Voltages_L3_L1_Voltage;
PQVoltageData.ar_LineVoltage[0] 			:= (EL3453.MDP5001_341_Input.Total_L_L_Voltages_L1_L2_Voltage + EL3453.MDP5001_341_Input.Total_L_L_Voltages_L2_L3_Voltage + EL3453.MDP5001_341_Input.Total_L_L_Voltages_L3_L1_Voltage) / 3;
PQVoltageData.ar_PowerFactor[1] 			:= EL3453.MDP5001_341_Input.L1_Power_Power_Factor;
PQVoltageData.ar_PowerFactor[2] 			:= EL3453.MDP5001_341_Input.L2_Power_Power_Factor;
PQVoltageData.ar_PowerFactor[3] 			:= EL3453.MDP5001_341_Input.L3_Power_Power_Factor;
PQVoltageData.ar_PowerFactor[0] 			:= EL3453.MDP5001_341_Input.Total_Basic_Power_Factor;
PQVoltageData.ar_current[1]					:= EL3453.MDP5001_341_Input.L1_Basic_Current;
PQVoltageData.ar_current[2]					:= EL3453.MDP5001_341_Input.L2_Basic_Current;
PQVoltageData.ar_current[3]					:= EL3453.MDP5001_341_Input.L3_Basic_Current;
PQVoltageData.ar_current[4]					:= EL3453.MDP5001_341_Input.Total_Basic_Neutral_Line_Current;
PQVoltageData.ar_Current[0]					:= (EL3453.MDP5001_341_Input.L1_Basic_Current + EL3453.MDP5001_341_Input.L2_Basic_Current + EL3453.MDP5001_341_Input.L3_Basic_Current) / 3;
PQVoltageData.ar_activePower[1]				:= EL3453.MDP5001_341_Input.L1_Power_Fundamental_active_Power_Fund;
PQVoltageData.ar_activePower[2]				:= EL3453.MDP5001_341_Input.L2_Power_Fundamental_active_Power_Fund;
PQVoltageData.ar_activePower[3]				:= EL3453.MDP5001_341_Input.L3_Power_Fundamental_active_Power_Fund;
PQVoltageData.ar_activePower[0]				:= EL3453.MDP5001_341_Input.Total_active_Fundamental_active_Power_Fund;
PQVoltageData.ar_ReactivePower[1]			:= EL3453.MDP5001_341_Input.L1_Power_Fundamental_Reactive_Power_Fund;
PQVoltageData.ar_ReactivePower[2]			:= EL3453.MDP5001_341_Input.L2_Power_Fundamental_Reactive_Power_Fund;
PQVoltageData.ar_ReactivePower[3]			:= EL3453.MDP5001_341_Input.L3_Power_Fundamental_Reactive_Power_Fund;
PQVoltageData.ar_ReactivePower[0]			:= EL3453.MDP5001_341_Input.Total_Reactive_Fundamental_Reactive_Power_Fund;
PQVoltageData.ar_ApparentPower[1]			:= EL3453.MDP5001_341_Input.L1_Power_Apparent_Power;
PQVoltageData.ar_ApparentPower[2]			:= EL3453.MDP5001_341_Input.L2_Power_Apparent_Power;
PQVoltageData.ar_ApparentPower[3]			:= EL3453.MDP5001_341_Input.L3_Power_Apparent_Power;
PQVoltageData.ar_ApparentPower[0]			:= EL3453.MDP5001_341_Input.Total_Apparent_Apparent_Power;
PQVoltageData.r_VoltageUnbalance			:= EL3453.MDP5001_341_Input.Total_Advanced_Voltage_Unbalance;
PQVoltageData.r_CurrentUnbalance			:= LineUnbalance(EL3453.MDP5001_341_Input.L1_Basic_Current, EL3453.MDP5001_341_Input.L2_Basic_Current, EL3453.MDP5001_341_Input.L3_Basic_Current);
PQVoltageData.ar_CurrentTHD[1]				:= EL3453.MDP5001_341_Input.L1_Advanced_Current_Total_Harmonic_Distortion;
PQVoltageData.ar_CurrentTHD[2]				:= EL3453.MDP5001_341_Input.L2_Advanced_Current_Total_Harmonic_Distortion;
PQVoltageData.ar_CurrentTHD[3]				:= EL3453.MDP5001_341_Input.L3_Advanced_Current_Total_Harmonic_Distortion;
PQVoltageData.ar_CurrentTHD[0]				:= EL3453.MDP5001_341_Input.Total_Advanced_Max_Current_Harmonic_Distortion;
PQVoltageData.ar_VoltageTHD[1]				:= EL3453.MDP5001_341_Input.L1_Advanced_Voltage_Total_Harmonic_Distortion;
PQVoltageData.ar_VoltageTHD[2]				:= EL3453.MDP5001_341_Input.L2_Advanced_Voltage_Total_Harmonic_Distortion;
PQVoltageData.ar_VoltageTHD[3]				:= EL3453.MDP5001_341_Input.L3_Advanced_Voltage_Total_Harmonic_Distortion;
PQVoltageData.ar_VoltageTHD[0]				:= EL3453.MDP5001_341_Input.Total_Advanced_Max_Voltage_Harmonic_Distortion;
PQVoltageData.ar_Frequency[1] 				:= ValueConversion(DataSelector._F, EL3453.MDP5001_341_Input.L1_Classic_Frequency);
PQVoltageData.ar_Frequency[2] 				:= ValueConversion(DataSelector._F, EL3453.MDP5001_341_Input.L2_Classic_Frequency);
PQVoltageData.ar_Frequency[3] 				:= ValueConversion(DataSelector._F, EL3453.MDP5001_341_Input.L3_Classic_Frequency);
PQVoltageData.ar_Frequency[0]				:= EL3453.MDP5001_341_Input.Total_Basic_Frequency;
PQVoltageData.r_EnergyConsumed				:= TO_REAL(EL3453.MDP5001_341_Input.Total_Active_Active_Negative_Energy)/1000;
PQVoltageData.r_EnergySupplied				:= TO_REAL(EL3453.MDP5001_341_Input.Total_Active_Active_Positive_Energy)/1000;
END_METHOD

METHOD ValueConversion : REAL
VAR_INPUT
	selector		: DataSelector;
	IN				: LINT;
END_VAR

VAR
	totalRatio		: REAL;
	scale			: REAL;
END_VAR
scale := 0.001; //default

CASE selector OF
 	DataSelector._C:
		totalRatio := CRatio;
	DataSelector._V:
		totalRatio := VRatio;
	DataSelector._P, DataSelector._Q:
		totalRatio := CRatio * VRatio * SEL(CInverse, 1, -1) / 1000;
	DataSelector._S, DataSelector._E:
		totalRatio := CRatio * VRatio / 1000;
	DataSelector._F:
		totalRatio := 1;
END_CASE

ValueConversion := TO_REAL(IN) * scale * totalRatio;
END_METHOD

END_FUNCTION_BLOCK

// ---- POUs/Functions-FBs-Programs/_acFunctions/AcPhasesOK.TcPOU
FUNCTION AcPhasesOK : BOOL
VAR_INPUT
	LineVoltageL1		: REAL;
	LineVoltageL2		: REAL;
	LineVoltageL3		: REAL;
END_VAR
VAR
	L1OK				: BOOL;
	L2OK				: BOOL;
	L3OK 				: BOOL;
END_VAR

L1OK := LIMIT(settings.GridParams.r_GridVoltageMin, LineVoltageL1, settings.GridParams.r_GridVoltageMax) = LineVoltageL1;
L2OK := LIMIT(settings.GridParams.r_GridVoltageMin, LineVoltageL2, settings.GridParams.r_GridVoltageMax) = LineVoltageL2;
L3OK := LIMIT(settings.GridParams.r_GridVoltageMin, LineVoltageL3, settings.GridParams.r_GridVoltageMax) = LineVoltageL3;


AcPhasesOK := L1OK AND L2OK AND L3OK;

END_FUNCTION

// ---- POUs/Functions-FBs-Programs/_acFunctions/LineUnbalance.TcPOU
FUNCTION LineUnbalance : REAL
VAR_INPUT
	r_L1		: REAL;
	r_L2		: REAL;
	r_L3		: REAL;
END_VAR
VAR
	r_Lavg		: REAL;
	r_dev1		: REAL;
	r_dev2		: REAL;
	r_dev3		: REAL;
	r_devMax	: REAL;
END_VAR

r_Lavg := (r_L1 + r_L2 + r_L3) / 3;

r_Dev1 := ABS(r_L1-r_Lavg);
r_Dev2 := ABS(r_L2-r_Lavg);
r_Dev3 := ABS(r_L3-r_Lavg);

r_devMax := MAX(r_Dev1, r_Dev2, r_Dev3);

LineUnbalance := r_devMax / MAX(r_Lavg,1) * 100;

END_FUNCTION

// ---- POUs/Objects/InternalPowerSupply/FB_InternalPowerSupply.TcPOU
FUNCTION_BLOCK FB_InternalPowerSupply implements itf_standardFB

VAR
	IO									: FB_InternalPowerSupply_IO;
	UPS									: FB_UPS;
	InternalPowerDemand					: ST_InternalPowerSupply_PowerDemand;
	b_EMStopActive 						: BOOL := FALSE;
	b_killUPS							: BOOL := FALSE;	
	b_HVDCAllowed						: BOOL;
	
	rtrig_CEEConnected					:	r_trig;
	LowBatShutdownTimer					:	TON;
	
	UPSChargeMode	:	bool;
END_VAR

VAR_IN_OUT CONSTANT
	st_params							: 	ST_InternalPowerSupply_Params;
END_VAR

VAR_INPUT
	st_CoolingDemandSupply				: ST_InternalPowerSupply_PowerDemand;
	st_PowerstackDemandSupply			: ST_InternalPowerSupply_PowerDemand;
	st_ACDCChargerDemandSupply			: ST_InternalPowerSupply_PowerDemand;
	st_DCBusDemandSupply				: ST_InternalPowerSupply_PowerDemand;
	
	b_BusbarACAvailable					: BOOL	:=	FALSE;
	e_BMSPowerstate						: eHVDC_Powerstatus;
	b_ConditioningOnBatteryAllowed		:	BOOL;
END_VAR

VAR_OUTPUT
	Get									: ST_InternalPowerSupply_Get;
	b_HVDC_Enable						: BOOL;
	b_PowerStackACRequired				: BOOL;
END_VAR


var
	b_ACPSU_OK				at %i* :	Bool;
	b_DCPSU_OK				at %i* :	Bool;
	b_CEEInputAvailable		AT %i* : 	Bool;
	b_enableHVDCPSU			AT %Q* :	Bool;
END_VAR

// call functions
UPS(b_24v_available := get.b_24VdcAvailable, st_params := st_params);
	get.UPS REF= UPS.Get;

ACPowerControl(st_params:=st_params, get:=get);
DCPowerControl(st_params:=st_params, b_UPSDemand24VDC := ups.b_UPSDemand24VDC,  get:= get);
HVDCPowerControl(enable := b_HVDCAllowed);

//if ups battery low warning occurs and no 24V is available, charging request failed and the system shuts down.
//If the system is connected to a source (HVDC, CEE, powerlock or internal AC), this is skipped.
//In that case, LowBatteryError will trip a system shutdown
LowBatShutdownTimer(in := UPS.Get.Events.b_BatteryLowWarning AND NOT get.b_24VdcAvailable, PT := st_params.LowBatteryShutdownTimer);
IF LowBatShutdownTimer.Q THEN
	SystemShutdown(TRUE);
END_IF

METHOD PRIVATE ACPowerControl : BOOL
VAR_IN_OUT CONSTANT
	st_params			: ST_Internalpowersupply_params;
END_VAR
VAR_IN_OUT
	get					: ST_InternalPowersupply_get;
END_VAR

VAR_INST
	tof_PowerstackACOffDelay: Tof := (PT := T#10S);
	ton_ACStartupDelay: TON;
	

END_VAR
//if cooling requires 400V, ask powerstack to supply either Main AC or inverter AC.
tof_PowerstackACOffDelay(IN := st_CoolingDemandSupply.b_Demand_400V and b_ConditioningOnBatteryAllowed);
b_PowerStackACRequired := tof_PowerstackACOffDelay.Q;

//after startup delay, internal 400VAC is available
ton_ACStartupDelay(IN := b_BusbarACAvailable, PT:=INT_TO_TIME(st_params.i_ACStartupDelay));
get.b_400VACAvailable := ton_ACstartupDelay.Q;

get.CEEInputActive := b_CEEInputAvailable;
END_METHOD

METHOD DCPowerControl : BOOL
VAR_IN_OUT CONSTANT
	st_params		: ST_Internalpowersupply_params;
	b_UPSDemand24VDC : BOOL;
END_VAR
VAR_IN_OUT
	get				: ST_Internalpowersupply_get;
END_VAR

VAR_INST
	ton_DCPSUStartupDelay: TON;
	ton_ACPSUStartupDelay: TON;
	tof_HVEnableOnUPSBattFailure	:	Tof := (pt := T#10M);
END_VAR
VAR
	DC_Required: BOOL;
END_VAR

ton_DCPSUStartupDelay(IN := get.b_HVDCAvailable, PT:= INT_TO_TIME(st_params.i_DCPSU_StartupDelay));
ton_ACPSUStartupDelay(IN := get.CEEInputActive, PT:= INT_TO_TIME(st_params.i_ACPSU_StartupDelay));

//if psu is not online after the startup delay, raise the fault status.
get.Events.b_ACPSUFault := ton_ACPSUStartupDelay.Q AND NOT b_ACPSU_OK;
get.Events.b_DCPSUFault := ton_DCPSUStartupDelay.Q AND NOT b_DCPSU_OK;

//if CEE psu has no status output, determine based on ups input and CEE AC detection
//	if not UPS.Get.BatteryTestActive then
//		DCPSU_OK := (get.UPS.r_InputVoltage > 20 and get.CEEInputActive);
//	end_if

//if CEE psu has status output, but no ac detection is present. Base AC detection on PSU output.
//get.CEEInputAvailable := DCPSU_OK or main_fast.AcDcCharger.Get.ACDetected;

//if any of the psu's is online, 24V is available
get.b_24VdcAvailable := b_ACPSU_OK OR b_DCPSU_OK;

//if no 400VAC available during 24VDC request, request HVDC ON for LVDC power				
internalPowerDemand.b_Demand_HVDC := NOT get.CEEInputActive AND b_DCPSU_OK;
END_METHOD

METHOD PUBLIC EMstop : BOOL

VAR_INST
	ton_HVDCShutdownTimeout	:	TON := (PT := T#5s);
END_VAR
//return true if done
b_EMStopActive := TRUE;

ton_HVDCShutdownTimeout(in:= get.b_HVDCAvailable);

//if HVDC shutdown takes too long, kill internal HVDC supply to 
get.Events.b_HVDCShutdownTimeExceeded := ton_HVDCShutdownTimeout.Q;

b_HVDCAllowed := FALSE;
//return true when all supplies are lost.
EMStop := NOT(get.b_HVDCAvailable);
END_METHOD

METHOD GetDiagnostics 
VAR_IN_OUT
	AddError		: ARRAY [*] OF FB_AddErrorST;
	a_ActiveEvents	: ARRAY [*] OF ST_ErrorStruct;
	w_Index			: WORD;
END_VAR
//check if this call works:
UPS.GetDiagnostics(AddError := AddError, a_ActiveEvents := a_ActiveEvents, w_Index := w_Index);
 
(*IPS*)
	(*AC PSU fault*)		AddError[w_Index](
			b_ErrorTrig			:= Get.Events.b_ACPSUFault,
			out_ST_Error			:= a_ActiveEvents[w_Index],
			w_ErrorID					:= 1,
			e_objectID				:= eObject_ID.InternalPowerSupply,
			s_Message				:= 'AC PSU fault',
			e_sev					:= eSeverity.Warning,
			t_triggerTime			:= T#3S,
			b_AutoClear			:= TRUE
			);
		w_Index := w_Index +1;
	(*DC PSU fault*)		AddError[w_Index](
			b_ErrorTrig			:= Get.Events.b_DCPSUFault,
			out_ST_Error			:= a_ActiveEvents[w_Index],
			w_ErrorID					:= 2,
			s_Message				:= 'DC PSU fault',
			e_sev					:= eSeverity.Warning,
			t_triggerTime			:= T#3S,
			b_AutoClear			:= TRUE
			);
		w_Index := w_Index +1;
	(*24V fault*)		AddError[w_Index](
			b_ErrorTrig			:= Get.Events.b_DCPSUFault AND Get.Events.b_ACPSUFault,
			out_ST_Error			:= a_ActiveEvents[w_Index],
			w_ErrorID					:= 3,
			s_Message				:= '24V supply failed',
			e_sev					:= eSeverity.QuickShutdown,
			);
		w_Index := w_Index +1;	
// 	(*CEE fuse tripped*)		AddError[w_Index](
// 			b_ErrorTrig			:= Get.Events.b_CEEInputFuseTripped,
// 			out_ST_Error			:= a_ActiveEvents[w_Index],
// 			w_ErrorID					:= 4,
// 			s_Message				:= 'CEE Standby power input fuse error',
// 			e_sev					:= eSeverity.Warning,
// 			b_AutoClear			:= TRUE,
// 			);
// 		w_Index := w_Index +1;
	(*internal grid fuse fault*)		AddError[w_Index](
			b_ErrorTrig		:= Get.Events.b_GridInputFuseTripped,
			out_ST_Error			:= a_ActiveEvents[w_Index],
			w_ErrorID					:= 5,
			s_Message				:= 'Internal supply Grid fuse error',
			e_sev					:= eSeverity.QuickShutdown,
			);
		w_Index := w_Index +1;
		
	(*EMSTOP HVDC shutdown failed*)		AddError[w_Index](
			b_ErrorTrig			:= Get.Events.b_HVDCShutdownTimeExceeded,
			out_ST_Error			:= a_ActiveEvents[w_Index],
			w_ErrorID					:= 6,
			s_Message				:= 'HVDC shutdown sequence failed',
			e_sev					:= eSeverity.QuickShutdown,			//<-- already in emstop, but this is a severe error
			);
		w_Index := w_Index +1;
		
	//Warnings
	(*UPS drained during operation*)		AddError[w_Index](
			b_ErrorTrig				:= UPS.Get.Events.b_BatteryLowWarning,
			out_ST_Error			:= a_ActiveEvents[w_Index],
			w_ErrorID				:= 8,
			s_Message				:= Concat('System shut down in: ', TO_STRING(LowBatShutdownTimer.PT - LowBatShutdownTimer.ET)),
			e_sev					:= eseverity.Warning,
			b_AutoClear				:= TRUE
			);
		w_Index := w_Index +1;
		
	//Warnings
	(*UPS battery low while on battery, initiate shutdown*) 	AddError[w_Index](
			b_ErrorTrig				:= LowBatShutdownTimer.Q,
			out_ST_Error			:= a_ActiveEvents[w_Index],
			w_ErrorID				:= 9,
			s_Message				:= 'Shutdown initiated: Halt system operation',
			e_sev					:= eseverity.QuickShutdown,
			b_AutoClear				:= TRUE
			);
		w_Index := w_Index +1;
END_METHOD

METHOD GetWearCounters : BOOL
VAR_INST
	ACPsuPoH				:	FB_Varlogger;
	DCPsuPoh				:	FB_Varlogger;
END_VAR

ACPsuPoH(				TriggerInput := IO.ACPSU_OK, 
						LogItemGroup :=  eLogItemGroupID.InternalPowerSupply, 
						LogItemName := 'AcPsuHrs', 
						LogType := eLogTypes.TrackOnTime);

DCPsuPoh(				TriggerInput := io.DCPSU_OK, 
						LogItemGroup :=  eLogItemGroupID.InternalPowerSupply, 
						LogItemName := 'DcPsuHrs', 
						LogType := eLogTypes.TrackOnTime);	

UPS.getWearCounters();
END_METHOD

METHOD HVDC_disable : BOOL;
b_HVDCAllowed := FALSE;
HVDC_disable := NOT b_HVDC_Enable;
END_METHOD

METHOD HVDC_Enable : BOOL
VAR_INPUT
END_VAR
b_HVDCAllowed := True;
END_METHOD

METHOD PRIVATE HVDCPowerControl : BOOL

VAR_INPUT
	enable		: BOOL;
END_VAR

VAR_INST
	TON_HVONDelay : TON := (PT := T#1S);
	TOF_HVOnDelay : TOF := (PT := T#1S);
END_VAR
//The powerstack demands HVDC directly. 
TOF_HVOnDelay(in:=	st_powerstackdemandsupply.b_Demand_HVDC OR 
					InternalPowerDemand.b_Demand_HVDC or 
					st_DCBusDemandSupply.b_Demand_HVDC or 
					st_ACDCChargerDemandSupply.b_Demand_HVDC or
					st_CoolingDemandSupply.b_Demand_HVDC);
b_HVDC_Enable := TOF_HVOnDelay.Q AND NOT b_EMStopActive AND enable;


TON_HVONDelay(in:= e_BMSPowerstate = eHVDC_Powerstatus.ON);
IF TON_HVONDelay.Q THEN
	IO.b_DCPsuEnable := TRUE;
	get.b_HVDCAvailable := TRUE;
ELSE
	IO.b_DCPsuEnable := FALSE;
	get.b_HVDCAvailable := FALSE;
END_IF
END_METHOD

{warning 'Add method implementation '}
METHOD Init : BOOL
END_METHOD

METHOD Reset : BOOL
//reset system
b_EMStopActive := FALSE;
get.Events.b_HVDCShutdownTimeExceeded := FALSE;
b_HVDCAllowed := TRUE;

Reset := NOT get.Events.b_GridInputFuseTripped;
//return true if ok
END_METHOD

METHOD SystemShutdown : BOOL

VAR_INPUT
	TimedShutdown		:	BOOL;
END_VAR

IF NOT TimedShutdown THEN
	get.Events.b_CEEPreventsShutdown := b_CEEInputAvailable;
	b_enableHVDCPSU	:= false;
	UPS.Shutdown();
END_IF
END_METHOD

END_FUNCTION_BLOCK

// ---- POUs/Objects/InternalPowerSupply/FB_InternalPowerSupply_IO.TcPOU
FUNCTION_BLOCK FB_InternalPowerSupply_IO

VAR_INPUT 
	b_DCPsuEnable		AT %Q* : BOOL := FALSE;
	b_ACPsuEnable		AT %Q* : BOOL := TRUE;
END_VAR

VAR_OUTPUT
	DCPSU_OK 			AT %I*: BOOL;
	ACPSU_OK 			AT %I*: BOOL;
	GridFuseOK 			AT %I*: BOOL;
END_VAR

END_FUNCTION_BLOCK

// ---- POUs/Objects/InternalPowerSupply/UPS/FB_UPS.TcPOU
FUNCTION_BLOCK FB_UPS
VAR_IN_OUT CONSTANT
	st_params		: ST_InternalPowersupply_params;
END_VAR

VAR_INPUT
	b_24V_Available	:	BOOL;
	r_BMSsoc		: 	REAL;
	b_EMSTOP		: 	BOOL;		
END_VAR
VAR_OUTPUT
	Get	: ST_UPSGET;
	b_UPSDemand24VDC	: BOOL;
END_VAR
VAR
	DisableUPS			AT %Q* : BOOL;
	DisconnectUPSInput	At %Q* : Bool;
	UPSData				AT %I* : ST_UPSDATA;	
	InputTimer					: TON := (PT := TIME#1S);
	
	SR_SoCLowWarning: SR;
	RS_SocLowError	: RS;

	
	TON_MinimumChargeTime	:	TON := (pt := T#1H);
	
	r_Hysteresis	: REAL := 5;
END_VAR

VAR PERSISTENT
	OriginalBatteryCapacity :	REAL	:=	100;	//Ah
	//Capacity loss not yet implemented
	ActualBattCapacity		:	REAL	:=	100;
	RemainingCapacity 		:	REAL	:=	100;

	LastBatteryCalibrationDate	:	DT;	
	ui_UPSBatteryHealth			:	Uint;
END_VAR

get.Events.b_BatteryLowError := FALSE;
get.Events.b_BatteryLowWarning := FALSE;

//no need to call this FB from the main sequence
//This FB is controlled via the internal power supply
 
Get.r_BatteryVoltage 	:= TO_REAL(UPSData.ui_BatteryVoltage) / 1000;
Get.r_InputVoltage		:= TO_REAL(UPSData.ui_InputVoltage) / 1000;
Get.r_OutputVoltage		:= TO_REAL(UPSData.ui_OutputVoltage) / 1000;
Get.r_OutputCurrent		:= TO_REAL(UPSData.ui_OutputCurrent) / 1000;
Get.ui_SOC 				:= GetSOC();
 
RS_SocLowError(
	SET:= Get.ui_SOC  < st_params.usi_UPSBattLowErrorSOC AND get.b_SystemOnBattery, 
	RESET1:= Get.ui_SOC  > st_params.usi_UPSBattLowWarningSOC OR get.b_ChargerActive,
	Q1 => get.Events.b_BatteryLowError
	);
	
SR_SocLowWarning(
	SET1:= Get.ui_SOC  < st_params.usi_UPSBattLowWarningSOC AND get.b_SystemOnBattery,
	RESET:= Get.ui_SOC  > st_params.usi_UPSBattLowWarningSOC + r_hysteresis OR get.b_SystemOnDCInput,
	Q1 => get.Events.b_BatteryLowWarning
	);
	
TON_MinimumChargeTime(in:=get.b_ChargerActive);

////When info message, also request 24VDC	
//SR_RequestCharging(
//	SET1:= get.Events.b_BatteryLowInfo,
//	RESET:= (Get.ui_SOC  = 100),
//	Q1 => b_UPSDemand24VDC
//	);

b_UPSDemand24VDC := true; //always require ups charging from now on

//fill get struct
//if system is charging, disable low battery error. Wait for sufficient r_SOC before disabling the low battery warning
get.b_ChargerActive := UPSData.udi_StatusFunctions.5;
get.b_systemonBattery := UPSData.udi_StatusFunctions.2;
get.b_SystemOnDCInput := UPSData.udi_StatusFunctions.1;
 
IF get.r_BatteryVoltage < 16 THEN
	get.Events.b_NoBatteryError := TRUE;
ELSE 
	get.Events.b_NoBatteryError := FALSE;
END_IF
 
//UPS input voltage should be OK shortly after IPS 24V coming online. Otherwise there is a problem
InputTimer(in:= b_24V_Available);
get.Events.b_InputVoltageWarning := InputTimer.Q AND (Get.r_InputVoltage < 20);


get.ui_UPSBatteryHealth := ui_UPSBatteryHealth;
batterySelftest();

METHOD BatterySelfTest : BOOL
VAR_INPUT
END_VAR

VAR
	r_AverageCurrentDropCount : REAL;
	dt_NextCalibration	:	DT;
	UPSBattCalibrationRequired	:	bool;
END_VAR

var_inst
	CalibrationStep		:	Uint := 0;
	ton_500msTimer			:	Ton:= (PT := T#500ms);	
	
	r_Vfloat				:	real;
	r_VInitialDrop			:	real;
	r_AverageCurrentInitialDrop	:	Real;
	ui_AverageCurrentDropCount	:	uint;
	
	r_Vstart				:	real;
	r_VEnd					:	real;
	r_UPSBatteryEnergyLoss	:	real;
END_VAR

var_inst
	r_InitialDropResistance	:	real;
	r_steadyStateDropValue	:	real;
END_VAR
IF st_params.t_UPSBattSelfTestInterval > T#0S THEN
	dt_NextCalibration := LastBatteryCalibrationDate + st_params.t_UPSBattSelfTestInterval;
END_IF


(*BOTH ton_initialdroptimer and b_UPSBatteryCalibrationActive are not declared --> What must be done with it.*)
//ton_500msTimer(in := not ton_500msTimer.q and b_UPSBatteryCalibrationActive);
//ton_InitialDropTimer(in := DisconnectUPSInput);


case CalibrationStep of
	
	0:	//idle, do nothing
		DisconnectUPSInput := FALSE;
		if gvl.dt_SystemDateTime > DT_NextCalibration then
			CalibrationStep := 1;
		END_IF
		
	1:	//calibration requested, wait for circumstances to be correct
		IF r_BMSsoc > 30 AND get.ui_SOC > 90 AND get.b_SystemOnDCInput AND NOT b_EMSTOP THEN
			CalibrationStep := 2;
			get.events.b_UPSBatteryCalibrationActive := true;
			r_AverageCurrentInitialDrop := 0;
			ui_AverageCurrentDropCount	:=	0;
		END_IF
		
	2:	// Initialize calibration and perform instant drop test to indicate pack resistance
		r_Vfloat	:=	get.r_BatteryVoltage;
		DisconnectUPSInput := true;
		
		if ton_500msTimer.Q then
			r_AverageCurrentInitialDrop := r_AverageCurrentInitialDrop + get.r_OutputCurrent/10;
			ui_AverageCurrentDropCount := ui_AverageCurrentDropCount + 1;
			if r_AverageCurrentDropCount = 10 then
				r_InitialDropResistance := (r_Vfloat-get.r_BatteryVoltage)/max(0.1, r_AverageCurrentInitialDrop);
				r_UPSBatteryEnergyLoss := 0;
				r_Vstart := get.r_BatteryVoltage;
				CalibrationStep := 3;
			END_IF
		end_if
		
	3: // track steady state energy loss
		
		if ton_500msTimer.Q then	
			r_UPSBatteryEnergyLoss := r_UPSBatteryEnergyLoss + (get.r_OutputCurrent/7200);
			
			if r_UPSBatteryEnergyLoss >= OriginalBatteryCapacity * 0.02 then
				r_steadyStateDropValue := (r_Vstart - get.r_BatteryVoltage) / max(r_UPSBatteryEnergyLoss, 0.01);
				CalibrationStep := 4;
			END_IF
		end_if
		
	4: //Calibration done, reset system
		DisconnectUPSInput := FALSE;
		get.events.b_UPSBatteryCalibrationActive := false;
		LastBatteryCalibrationDate := gvl.dt_SystemDateTime;
		
		//a equivalent SOH calculation should be created here, based on InitialDropResistance and steadyStateDropValue
		
		CalibrationStep := 0;
END_CASE


//stop calibration if voltage drops to far.
if get.events.b_UPSBatteryCalibrationActive and get.r_BatteryVoltage < 24 then
	DisconnectUPSInput := FALSE;
	get.events.b_UPSBatteryCalibrationActive := false;
	LastBatteryCalibrationDate := gvl.dt_SystemDateTime;
	ui_UPSBatteryHealth := 1; //1% SOH as we cannot complete calibration
	CalibrationStep := 0;
END_IF
END_METHOD

METHOD GetDiagnostics 
VAR_IN_OUT
	AddError		: ARRAY [*] OF FB_AddErrorST;
	a_ActiveEvents	: ARRAY [*] OF ST_ErrorStruct;
	w_Index			: WORD;
END_VAR
(*UPS*)
	(*Low battery error*)		AddError[w_Index](
			b_ErrorTrig			:= Get.Events.b_BatteryLowError,
			out_ST_Error			:= a_ActiveEvents[w_Index],
			w_ErrorID					:= 1,
			e_objectID				:=	eObject_ID.UPS,
			s_Message				:= 'low battery error',
			e_sev					:= eSeverity.Normalshutdown,
			t_triggerTime			:= T#30S,
			);
		w_Index := w_Index +1;
	(*low battery warning*)		AddError[w_Index](
			b_ErrorTrig			:= Get.Events.b_BatteryLowWarning,
			out_ST_Error			:= a_ActiveEvents[w_Index],
			w_ErrorID					:= 2,
			s_Message				:= 'low battery warning',
			e_sev					:= eSeverity.warning,
			b_AutoClear				:= TRUE,
			t_triggerTime			:= T#1S,
			);
		w_Index := w_Index +1;
	(*UPS input undervoltage*)		AddError[w_Index](
			b_ErrorTrig			:= Get.Events.b_InputVoltageWarning,
			out_ST_Error			:= a_ActiveEvents[w_Index],
			w_ErrorID					:= 3,
			s_Message				:= 'UPS input undervoltage',
			e_sev					:= eSeverity.Warning,
			b_AutoClear				:= TRUE,
			);
		w_Index := w_Index +1;
	(*no UPS battery*)		AddError[w_Index](
			b_ErrorTrig		:= Get.Events.b_NoBatteryError,
			out_ST_Error			:= a_ActiveEvents[w_Index],
			w_ErrorID					:= 4,
			s_Message				:= 'no battery error',
			e_sev					:= eSeverity.Warning,
			t_triggerTime			:= T#5S,
			);
		w_Index := w_Index +1;
END_METHOD

METHOD GetSoC : USINT
VAR_INST
	ton_SOCUpdate			:	TON	:=	(PT := T#500MS);
	ton_TailCurrentTimer	:	TON;
	Ton_OverrideSocEmpty	:	ton	:=	(PT := T#1M);
	Ton_OverrideSocBelowHalfFull	:	ton	:=	(PT := T#1M);
	Ton_OverrideSocAboveHalfFull	:	ton	:=	(PT := T#1M);
	
	fTrig_ChargingDone				:	f_trig;

	CapacityLoss			:	REAL;

	RatedDischargeTime		:	REAL	:=	20; //hours
	ChargeEfficiency		:	REAL	:=	1;//0.95;
	PeukertExponent			:	REAL	:=	1.13;
	TailCurrentRate			:	REAL	:=	0.02;
	ChargedDetectionTime	:	TIME	:=	T#3M;
	
END_VAR
ton_SOCUpdate(in := NOT ton_SOCUpdate.Q);

fTrig_ChargingDone(clk := get.b_ChargerActive);
IF fTrig_ChargingDone.Q AND get.b_SystemOnDCInput THEN
	RemainingCapacity := ActualBattCapacity;
END_IF

	
	
IF ton_SOCUpdate.q THEN
	ton_TailCurrentTimer(in:= 	UPSData.ui_BatteryVoltage >= 28000 AND 
								UPSData.ui_BatteryChargingCurrent < ((OriginalBatteryCapacity*TailCurrentRate)*1000) AND
								get.b_ChargerActive
								, pt:= ChargedDetectionTime);	

	Ton_OverrideSocBelowHalfFull(in:= 	between(UPSData.ui_BatteryVoltage, 23000, 24000) AND get.b_systemonBattery);
	Ton_OverrideSocEmpty(in:= 			between(UPSData.ui_BatteryVoltage, 15000, 23000) AND get.b_systemonBattery); //added >15v check to prevent SOC override when ups data readout fails
	Ton_OverrideSocAboveHalfFull(in := 	UPSData.ui_BatteryVoltage > SEL(get.b_ChargerActive, 25000, 26000));
	//When fully charged, recalibrate AH.
	IF ton_TailCurrentTimer.Q THEN
		RemainingCapacity := ActualBattCapacity;
	END_IF
	
	IF Ton_OverrideSocAboveHalfFull.Q THEN
		 RemainingCapacity := LIMIT(50, RemainingCapacity, ActualBattCapacity); //SOC limited to 50% if voltage <24V
END_IF

	IF Ton_OverrideSocBelowHalfFull.Q THEN
		 RemainingCapacity := LIMIT(0, RemainingCapacity, ActualBattCapacity/2); //SOC limited to 50% if voltage <24V
	END_IF	

	IF Ton_OverrideSocEmpty.Q THEN
		 RemainingCapacity := 0;
	END_IF		

//basic lineaire r_SOC berekening voor nu
	RemainingCapacity := LIMIT(0, RemainingCapacity + (ChargeEfficiency*(TO_REAL(UPSData.ui_BatteryChargingCurrent)/1000)/7200), ActualBattCapacity);
//Undervoltage recalibration
		//charging
	CapacityLoss := 0;
	IF get.b_systemonBattery AND get.r_OutputCurrent > 0 THEN
		CapacityLoss := (get.r_OutputCurrent/EXPT(OriginalBatteryCapacity/(get.r_OutputCurrent*RatedDischargeTime), PeukertExponent-1))/7200;
	END_IF
	RemainingCapacity := LIMIT(0, RemainingCapacity - CapacityLoss, ActualBattCapacity);
		//23V is 0%
	END_IF

GetSoC := TO_USINT((RemainingCapacity/ActualBattCapacity)*100);
END_METHOD

METHOD GetWearCounters : BOOL
VAR_INST
	UpsOnBatt				:	FB_Varlogger;
	UPSBattLow				:	FB_Varlogger;
END_VAR

UpsOnBatt(				TriggerInput := get.b_SystemOnBattery, 
						LogItemGroup :=  eLogItemGroupID.InternalPowerSupply, 
						LogItemName := 'UpsOnBattHrs', 
						LogType := eLogTypes.TrackOnTime);

UPSBattLow(				TriggerInput := get.Events.b_BatteryLowWarning, 
						LogItemGroup :=  eLogItemGroupID.InternalPowerSupply, 
						LogItemName := 'UpsBattLowCnt', 
						LogType := eLogTypes.TrackCycles);
END_METHOD

{warning 'Add method implementation '}
METHOD Reset : BOOL
END_METHOD

METHOD Shutdown : BOOL


VAR_INST
	TP_EnableDelay	: TP := (PT:= T#500MS);
END_VAR
DisableUPS := TRUE;

//IF DisableUPS = FALSE THEN
//	TP_EnableDelay(IN:= TRUE);
//END_IF

//TON_EnableDelay(IN:= NOT DisableUPS);
//IF TON_DisablePulse.Q THEN
//	DisableUPS := FALSE;
//END_IF
END_METHOD

END_FUNCTION_BLOCK

// ---- POUs/Objects/BMS/FB_BMS.TcPOU
FUNCTION_BLOCK FB_BMS
VAR PERSISTENT
	ui_CycleCount				: UINT;
	r_CumDischargeEnergy		: REAL; // kWh
	r_CumChargeEnergy			: REAL; // kWh
	r_maxVoltageEver	 		: REAL;
	r_maxChargeCurrentEver		: REAL;
	r_maxDischargeCurrentEver	: REAL;
	dt_LastCalibrationDate		: DT;
END_VAR

VAR_IN_OUT CONSTANT
	st_params	: st_BMS_Params;
END_VAR

VAR_IN_OUT
 	st_service	: st_BMS_service;
END_VAR

VAR_OUTPUT
	PowerStatus: eHVDC_Powerstatus := 0;
END_VAR
VAR_INPUT
	Set 					: st_BMS_Set;
	b_HVDCEnable			: BOOL;
	by_NoOfStrings			: BYTE;
END_VAR

VAR_OUTPUT
	get						: st_BMS_Get;
	b_InternalHVDCAllowed	:	BOOL;
END_VAR

VAR	
	InitDone			:	Bool := false;
	b_HVDC_OnRq			: BOOL;	
	FBState					:	ePOUState;
	IO					:	FB_BMS_IO;
	InitTimeout			: 	TON := (PT:=T#3S);
	BMS_24V_StartupTimer : TON := (PT := TIME#2S0MS);
	
	DeviceIDcounter		: WORD;
	
	//SFC
	SFCInit				: BOOL := FALSE;
	SFCReset			: BOOL := FALSE;
	
	//Modbus
	b_MBComErrorActive	: 	BOOL 	:= FALSE;
	ComTimer			:	Ton := (PT := TIME#100MS);
	t_TimeOut			: 	TIME := T#500MS;
	
	ResetBMS	:	Bool; 
	b_BMSShutdownRequested: BOOL;
	
	BMSReadIntervalTimer	 : TON := (PT := TIME#1S0MS);
	
	b_ManualReset	:BOOL;
	BMSDataValid		:	Bool;
	
	arDatalogMBMU	: ARRAY [0..58] OF WORD;
	arDatalogSBMU	: ARRAY[0..3] OF ARRAY[0..55] OF WORD;
	ARDatalogEMS	: ARRAY [0..16] OF WORD;
	
	AutoSOCCalibrationRequired	:	Bool;
END_VAR

VAR CONSTANT
	e_ID 				: eObject_ID := eObject_ID.Battery;
END_VAR

BMSDatalogger(b_enable := InitDone);
(*
FB_BMS

Inputs
	Set.b_EnableBMS				:	BOOL;
		Start BMS SFC sequence and initializes BMS. False means full BMS powerdown, so no status logging.
		With HVDC enabled, setting this value to False has no effect. Only after HVDC powerdown this value is tested.
		
	Set.b_ClearFault				:	BOOL;
		Clear errors and warning in BMS system. Set to true to initiate reset. Value resets automatically to false.
	
	Set.b_HVDC_Required			: 	BOOL;
		Set by FB_internalPowersupply. True initiates and keeps HVDC on, False initiates and retains powerdown

Outputs
	BMSGET
		-Some general status info
		-BATTinfo	struct with main operation battery data
		-MBMU_Status 	struct with detailed MBMU data
		-SBMU			Struct with detailed data per SBMU
		-Events			Warnings & Errors as per Sunspec list.
*)

IF InitDone THEN
	//INIT step
	//b_MBComErrorActive := FALSE;
	
	//CALL methods/functions
	//Link MBMU data when appropriate
	GetBatteryInfo(in := get.MBMU.BatteryStatus, OUT:= get.BatteryInfo);
	
	IF st_params.b_EnableAutoCalibration THEN
		IF dt_LastCalibrationDate > gvl.dt_SystemDateTime OR 
			(dt_LastCalibrationDate + st_params.T_AutoCalibrationInterval) < gvl.dt_SystemDateTime THEN
			get.T_RemainingTimeToAutoCalibration := T#0S;
			AutoSOCCalibrationRequired := TRUE;
		ELSE
			AutoSOCCalibrationRequired := FALSE;
			get.T_RemainingTimeToAutoCalibration := (dt_LastCalibrationDate + st_params.T_AutoCalibrationInterval) - gvl.dt_SystemDateTime;
		END_IF
	ELSE
		AutoSOCCalibrationRequired := FALSE;
		get.T_RemainingTimeToAutoCalibration := ST_Params.t_AutoCalibrationInterval;
	END_IF

		
	

	//get.LastCalibrationTime := dt_LastCalibrationDate;
	
	IF get.BatteryInfo.r_SOC < st_params.r_InternalConditioningSoCMin OR get.BatteryInfo.ar_CellVoltage[eSubValues.Minimum] < 3 THEN
		b_InternalHVDCAllowed := FALSE;
	ELSE
		b_InternalHVDCAllowed := TRUE;
	END_IF
	
	IO();
	
	BMSReadIntervalTimer(in:= not BMSReadIntervalTimer.Q);
	
	//Reset ErrorActive before entering SFC. 
	//any remaining error in the Modbus methods will set Erroractive again. 
	//This is pushed to events in BMS_Diagnostics
	
	//TEMPBMSHB();
	//hv required not allowed if BMS not enabled
	IF set.b_enable AND FBstate <> epoustate.EMSTOP THEN
		b_HVDC_OnRq := b_HVDCEnable OR st_params.b_forcePrecharging;
		
	ELSE
		b_HVDC_OnRq := FALSE;	
	END_IF
	
	//shutdown allowed if hvdc is offline
	b_BMSShutdownRequested := (NOT Set.b_Enable) AND get.MBMU.BatteryStatus.e_BMS_PowerOnStatus <> ePowerOnStatus.On; 
	
	IF b_ManualReset THEN
		Reset();
	END_IF
	
	//SFC delayed pulse trigger
	BMSSFC();
	
	BMS_Diagnostics();
	
	BMSDataValid := ((NOT get.Events.b_COMMUNICATION_ERROR) AND NOT (get.BatteryInfo.e_BMS_Status = eBMS_Status.Init));
END_IF

ACTION aBMSPoweroff:
IO.b_BMSEnable := FALSE;

get.BatteryInfo.b_BMSHeartBeatOK := FALSE;
get.BatteryInfo.e_BMS_PowerOnStatus := ePowerOnStatus.Off;
get.BatteryInfo.e_BMS_Status := eBMS_Status.Off;

get.MBMU.BatteryStatus.b_BMSHeartBeatOK := FALSE;
get.MBMU.BatteryStatus.e_BMS_PowerOnStatus := ePowerOnStatus.Off;
get.MBMU.BatteryStatus.e_BMS_Status := eBMS_Status.Off;

FBState := ePOUState.OFF;
END_ACTION

ACTION aBMSPowerOn:

//230V inverter requires some startup time. Start this first to init SBMU before MBMU
//This may not be needed, but the idea is to make sure the MBMU can reach the SBMU's at boot.
FBState := ePOUState.PowerUp;
io.b_BMSEnable := TRUE;
BMS_24V_StartupTimer(IN:=io.b_BMSEnable);
END_ACTION

ACTION aClearFaults:
SFCTip := ClearBMSFaults(st_params);
END_ACTION

ACTION aDisableInsulationMonitor:
SFCTip := OpenInsulationSwitch(st_params, TRUE);
END_ACTION

ACTION aGetMBMUData:
SFCTip := GetMBMUData(st_params);
END_ACTION

ACTION aGetSBMUData:
SFCTip := GetSBMUData(st_params);
END_ACTION

ACTION aGetStaticData:

IF (DeviceIDcounter=0) THEN
	IF GetMBMUStaticSystemData(st_params) THEN
		DeviceIDcounter:=1;
	END_IF;
ELSE
	IF GetSBMUStaticSystemData(st_params, DeviceIDcounter) THEN
		DeviceIDcounter := DeviceIDcounter+1;
	END_IF
	
	IF DeviceIDcounter > by_NoOfStrings THEN//BMSGet.MBMU_Status.by_NumberOfSubSystems THEN
		DeviceIDcounter:=0;
		SFCtip := NOT SFCtip;
	END_IF
END_IF
END_ACTION

ACTION aGetStatus:
IF GetSystemStatus(st_params) THEN
	IF FBState = ePOUState.PowerUp THEN FBState := ePOUState.Init; END_IF
	SFCtip := NOT SFCtip;
END_IF
END_ACTION

ACTION aInit:
DeviceIDcounter := 0;
SFCReset := FALSE;
b_MBComErrorActive := FALSE;
END_ACTION

ACTION aSetDateTime:
SFCTip := SetBMSDateTime(st_params);
END_ACTION

ACTION aSetPowerMode:
SFCTip := SetPowerMode(st_params);
END_ACTION

ACTION aWatchdog:
IF FBState = ePOUState.Init THEN FBState := ePOUState.Normal; END_IF

SFCtip := BMSHeartBeat(st_params);
DeviceIDcounter := 0;
END_ACTION

METHOD PRIVATE BMS_Diagnostics : BOOL
VAR
	
END_VAR

